LIN {X 0,Y 532.067,Z 647.363,A -85,B 0,C 180,E1 -4293.412,E2 -4293.412} C_VEL
LIN {X 0,Y 531.8,Z 656.616,A -85,B 0,C 180,E1 -4294.144,E2 -4294.144} C_VEL
LIN {X 0,Y 531.496,Z 665.466,A -85,B 0,C 180,E1 -4294.968,E2 -4294.968} C_VEL
LIN {X 0,Y 531.231,Z 673.986,A -85,B 0,C 180,E1 -4295.9,E2 -4295.9} C_VEL
LIN {X 0,Y 531.025,Z 681.116,A -85,B 0,C 180,E1 -4296.813,E2 -4296.813} C_VEL
LIN {X 0,Y 530.872,Z 687.423,A -85,B 0,C 180,E1 -4297.752,E2 -4297.752} C_VEL
LIN {X 0,Y 530.706,Z 693.662,A -85,B 0,C 180,E1 -4298.847,E2 -4298.847} C_VEL
LIN {X 0,Y 530.602,Z 698.519,A -85,B 0,C 180,E1 -4299.857,E2 -4299.857} C_VEL
LIN {X 0,Y 530.516,Z 703.385,A -85,B 0,C 180,E1 -4301.061,E2 -4301.061} C_VEL
LIN {X 0,Y 530.472,Z 707.261,A -85,B 0,C 180,E1 -4302.259,E2 -4302.259} C_VEL
LIN {X 0,Y 530.408,Z 709.397,A -85,B 0,C 180,E1 -4303.052,E2 -4303.052} C_VEL
LIN {X 0,Y 530.345,Z 712.263,A -85,B 0,C 180,E1 -4304.631,E2 -4304.631} C_VEL
LIN {X 0,Y 530.384,Z 713.236,A -85,B 0,C 180,E1 -4305.418,E2 -4305.418} C_VEL
LIN {X 0,Y 530.361,Z 713.956,A -85,B 0,C 180,E1 -4306.981,E2 -4306.981} C_VEL
LIN {X 0,Y 530.413,Z 713.28,A -85,B 0,C 180,E1 -4308.536,E2 -4308.536} C_VEL
LIN {X 0,Y 530.407,Z 712.529,A -85,B 0,C 180,E1 -4309.31,E2 -4309.31} C_VEL
LIN {X 0,Y 530.379,Z 709.752,A -85,B 0,C 180,E1 -4310.851,E2 -4310.851} C_VEL
LIN {X 0,Y 530.48,Z 706.779,A -85,B 0,C 180,E1 -4312.004,E2 -4312.004} C_VEL
LIN {X 0,Y 530.561,Z 702.949,A -85,B 0,C 180,E1 -4313.153,E2 -4313.153} C_VEL
LIN {X 0,Y 530.614,Z 698.263,A -85,B 0,C 180,E1 -4314.299,E2 -4314.299} C_VEL
LIN {X 0,Y 530.728,Z 692.661,A -85,B 0,C 180,E1 -4315.443,E2 -4315.443} C_VEL
LIN {X 0,Y 530.851,Z 685.927,A -85,B 0,C 180,E1 -4316.585,E2 -4316.585} C_VEL
LIN {X 0,Y 531.062,Z 679.305,A -85,B 0,C 180,E1 -4317.535,E2 -4317.535} C_VEL
LIN {X 0,Y 531.334,Z 671.548,A -85,B 0,C 180,E1 -4318.484,E2 -4318.484} C_VEL
LIN {X 0,Y 531.547,Z 662.423,A -85,B 0,C 180,E1 -4319.432,E2 -4319.432} C_VEL
LIN {X 0,Y 531.931,Z 652.624,A -85,B 0,C 180,E1 -4320.284,E2 -4320.284} C_VEL
LIN {X 0,Y 532.218,Z 642.253,A -85,B 0,C 180,E1 -4321.041,E2 -4321.041} C_VEL
LIN {X 0,Y 532.579,Z 629.489,A -85,B 0,C 180,E1 -4321.796,E2 -4321.796} C_VEL
LIN {X 0,Y 532.858,Z 615.986,A -85,B 0,C 180,E1 -4322.41,E2 -4322.41} C_VEL
LIN {X 0,Y 533.023,Z 602.545,A -85,B 0,C 180,E1 -4322.858,E2 -4322.858} C_VEL
LIN {X 0,Y 533.164,Z 588.82,A -85,B 0,C 180,E1 -4323.165,E2 -4323.165} C_VEL
LIN {X 0,Y 533.446,Z 541.847,A -85,B 0,C 180,E1 -4323.807,E2 -4323.807} C_VEL
LIN {X 0,Y 530.981,Z 534.347,A -85,B 0,C 180,E1 -4323.985,E2 -4323.985} C_VEL
LIN {X 0,Y 531.079,Z 534.333,A -85,B 0,C 180,E1 -4326.077,E2 -4326.077} C_VEL
LIN {X 0,Y 531.028,Z 534.337,A -85,B 0,C 180,E1 -4329.139,E2 -4329.139} C_VEL
LIN {X 0,Y 531.038,Z 534.335,A -85,B 0,C 180,E1 -4332.225,E2 -4332.225} C_VEL
LIN {X 0,Y 530.992,Z 534.346,A -85,B 0,C 180,E1 -4335.35,E2 -4335.35} C_VEL
LIN {X 0,Y 530.988,Z 534.339,A -85,B 0,C 180,E1 -4338.522,E2 -4338.522} C_VEL
LIN {X 0,Y 530.997,Z 534.34,A -85,B 0,C 180,E1 -4340.938,E2 -4340.938} C_VEL
LIN {X 0,Y 530.978,Z 534.34,A -85,B 0,C 180,E1 -4344.225,E2 -4344.225} C_VEL
LIN {X 0,Y 531.01,Z 534.336,A -85,B 0,C 180,E1 -4346.744,E2 -4346.744} C_VEL
LIN {X 0,Y 530.991,Z 534.345,A -85,B 0,C 180,E1 -4349.322,E2 -4349.322} C_VEL
LIN {X 0,Y 530.978,Z 534.337,A -85,B 0,C 180,E1 -4352.104,E2 -4352.104} C_VEL
LIN {X 0,Y 530.98,Z 534.339,A -85,B 0,C 180,E1 -4354.854,E2 -4354.854} C_VEL
LIN {X 0,Y 530.965,Z 534.346,A -85,B 0,C 180,E1 -4357.508,E2 -4357.508} C_VEL
LIN {X 0,Y 530.984,Z 534.339,A -85,B 0,C 180,E1 -4360.433,E2 -4360.433} C_VEL
LIN {X 0,Y 530.97,Z 534.348,A -85,B 0,C 180,E1 -4363.283,E2 -4363.283} C_VEL
LIN {X 0,Y 530.987,Z 534.341,A -85,B 0,C 180,E1 -4365.621,E2 -4365.621} C_VEL
LIN {X 0,Y 530.996,Z 534.338,A -85,B 0,C 180,E1 -4368.565,E2 -4368.565} C_VEL
LIN {X 0,Y 530.959,Z 534.346,A -85,B 0,C 180,E1 -4371.53,E2 -4371.53} C_VEL
LIN {X 0,Y 530.978,Z 534.343,A -85,B 0,C 180,E1 -4374.382,E2 -4374.382} C_VEL
LIN {X 0,Y 531.031,Z 534.438,A -85,B 0,C 180,E1 -4377.565,E2 -4377.565} C_VEL
LIN {X 0,Y 533.392,Z 545.862,A -85,B 0,C 180,E1 -4379.518,E2 -4379.518} C_VEL
LIN {X 0,Y 533.092,Z 562.113,A -85,B 0,C 180,E1 -4382.043,E2 -4382.043} C_VEL
LIN {X 0,Y 532.635,Z 581.906,A -85,B 0,C 180,E1 -4385.025,E2 -4385.025} C_VEL
LIN {X 0,Y 532.253,Z 602.681,A -85,B 0,C 180,E1 -4388.101,E2 -4388.101} C_VEL
LIN {X 0,Y 531.882,Z 623.757,A -85,B 0,C 180,E1 -4391.112,E2 -4391.112} C_VEL
LIN {X 0,Y 531.506,Z 643.326,A -85,B 0,C 180,E1 -4393.879,E2 -4393.879} C_VEL
LIN {X 0,Y 531.467,Z 651.526,A -85,B 0,C 180,E1 -4395.048,E2 -4395.048} C_VEL
LIN {X 0,Y 532.806,Z 661.786,A -85,B 0,C 180,E1 -4395.227,E2 -4395.227} C_VEL
LIN {X 0,Y 532.44,Z 759.968,A -85,B 0,C 180,E1 -4396.572,E2 -4396.572} C_VEL
LIN {X 0,Y 532.23,Z 773.227,A -85,B 0,C 180,E1 -4396.907,E2 -4396.907} C_VEL
LIN {X 0,Y 531.99,Z 785.378,A -85,B 0,C 180,E1 -4397.362,E2 -4397.362} C_VEL
LIN {X 0,Y 531.828,Z 796.691,A -85,B 0,C 180,E1 -4397.932,E2 -4397.932} C_VEL
LIN {X 0,Y 531.572,Z 807.906,A -85,B 0,C 180,E1 -4398.659,E2 -4398.659} C_VEL
LIN {X 0,Y 531.282,Z 818.538,A -85,B 0,C 180,E1 -4399.521,E2 -4399.521} C_VEL
LIN {X 0,Y 531.06,Z 828.119,A -85,B 0,C 180,E1 -4400.479,E2 -4400.479} C_VEL
LIN {X 0,Y 530.886,Z 835.964,A -85,B 0,C 180,E1 -4401.436,E2 -4401.436} C_VEL
LIN {X 0,Y 530.685,Z 843.624,A -85,B 0,C 180,E1 -4402.582,E2 -4402.582} C_VEL
LIN {X 0,Y 530.604,Z 850.682,A -85,B 0,C 180,E1 -4403.918,E2 -4403.918} C_VEL
LIN {X 0,Y 530.459,Z 855.372,A -85,B 0,C 180,E1 -4405.06,E2 -4405.06} C_VEL
LIN {X 0,Y 530.516,Z 858.961,A -85,B 0,C 180,E1 -4406.203,E2 -4406.203} C_VEL
LIN {X 0,Y 530.457,Z 860.811,A -85,B 0,C 180,E1 -4406.963,E2 -4406.963} C_VEL
LIN {X 0,Y 530.41,Z 862.199,A -85,B 0,C 180,E1 -4407.722,E2 -4407.722} C_VEL
LIN {X 0,Y 530.344,Z 863.787,A -85,B 0,C 180,E1 -4409.241,E2 -4409.241} C_VEL
LIN {X 0,Y 530.342,Z 864,A -85,B 0,C 180,E1 -4410,E2 -4410} C_VEL
LIN {X 0,Y 530.361,Z 863.183,A -85,B 0,C 180,E1 -4411.519,E2 -4411.519} C_VEL
LIN {X 0,Y 530.41,Z 862.195,A -85,B 0,C 180,E1 -4412.279,E2 -4412.279} C_VEL
LIN {X 0,Y 530.457,Z 860.807,A -85,B 0,C 180,E1 -4413.038,E2 -4413.038} C_VEL
LIN {X 0,Y 530.523,Z 857.895,A -85,B 0,C 180,E1 -4414.179,E2 -4414.179} C_VEL
LIN {X 0,Y 530.525,Z 853.948,A -85,B 0,C 180,E1 -4415.321,E2 -4415.321} C_VEL
LIN {X 0,Y 530.6,Z 848.259,A -85,B 0,C 180,E1 -4416.582,E2 -4416.582} C_VEL
LIN {X 0,Y 530.759,Z 841.231,A -85,B 0,C 180,E1 -4417.801,E2 -4417.801} C_VEL
LIN {X 0,Y 530.929,Z 832.99,A -85,B 0,C 180,E1 -4418.948,E2 -4418.948} C_VEL
LIN {X 0,Y 531.137,Z 824.534,A -85,B 0,C 180,E1 -4419.905,E2 -4419.905} C_VEL
LIN {X 0,Y 531.409,Z 814.088,A -85,B 0,C 180,E1 -4420.863,E2 -4420.863} C_VEL
LIN {X 0,Y 531.694,Z 803.35,A -85,B 0,C 180,E1 -4421.656,E2 -4421.656} C_VEL
LIN {X 0,Y 531.933,Z 792.394,A -85,B 0,C 180,E1 -4422.301,E2 -4422.301} C_VEL
LIN {X 0,Y 532.124,Z 780.764,A -85,B 0,C 180,E1 -4422.83,E2 -4422.83} C_VEL
LIN {X 0,Y 532.369,Z 767.341,A -85,B 0,C 180,E1 -4423.261,E2 -4423.261} C_VEL
LIN {X 0,Y 532.479,Z 754.056,A -85,B 0,C 180,E1 -4423.525,E2 -4423.525} C_VEL
LIN {X 0,Y 532.679,Z 659.294,A -85,B 0,C 180,E1 -4424.811,E2 -4424.811} C_VEL
LIN {X 0,Y 531.429,Z 651.372,A -85,B 0,C 180,E1 -4424.973,E2 -4424.973} C_VEL
LIN {X 0,Y 531.691,Z 634.591,A -85,B 0,C 180,E1 -4427.302,E2 -4427.302} C_VEL
LIN {X 0,Y 531.965,Z 611.61,A -85,B 0,C 180,E1 -4430.357,E2 -4430.357} C_VEL
LIN {X 0,Y 532.115,Z 589.217,A -85,B 0,C 180,E1 -4433.343,E2 -4433.343} C_VEL
LIN {X 0,Y 532.194,Z 568.689,A -85,B 0,C 180,E1 -4436.104,E2 -4436.104} C_VEL
LIN {X 0,Y 532.152,Z 547.238,A -85,B 0,C 180,E1 -4439.036,E2 -4439.036} C_VEL
LIN {X 0,Y 531.969,Z 539.363,A -85,B 0,C 180,E1 -4440.135,E2 -4440.135} C_VEL
LIN {X 0,Y 531.066,Z 534.337,A -85,B 0,C 180,E1 -4440.876,E2 -4440.876} C_VEL
LIN {X 0,Y 530.994,Z 534.339,A -85,B 0,C 180,E1 -4443.773,E2 -4443.773} C_VEL
LIN {X 0,Y 530.96,Z 534.346,A -85,B 0,C 180,E1 -4446.559,E2 -4446.559} C_VEL
LIN {X 0,Y 530.993,Z 534.339,A -85,B 0,C 180,E1 -4449.443,E2 -4449.443} C_VEL
LIN {X 0,Y 530.982,Z 534.343,A -85,B 0,C 180,E1 -4452.457,E2 -4452.457} C_VEL
LIN {X 0,Y 530.989,Z 534.339,A -85,B 0,C 180,E1 -4455.621,E2 -4455.621} C_VEL
LIN {X 0,Y 531.004,Z 534.343,A -85,B 0,C 180,E1 -4458.565,E2 -4458.565} C_VEL
LIN {X 0,Y 530.963,Z 534.342,A -85,B 0,C 180,E1 -4461.529,E2 -4461.529} C_VEL
LIN {X 0,Y 530.958,Z 534.348,A -85,B 0,C 180,E1 -4464.38,E2 -4464.38} C_VEL
LIN {X 0,Y 530.972,Z 534.343,A -85,B 0,C 180,E1 -4467.133,E2 -4467.133} C_VEL
LIN {X 0,Y 530.975,Z 534.341,A -85,B 0,C 180,E1 -4469.803,E2 -4469.803} C_VEL
LIN {X 0,Y 531.02,Z 534.344,A -85,B 0,C 180,E1 -4472.467,E2 -4472.467} C_VEL
LIN {X 0,Y 531.011,Z 534.34,A -85,B 0,C 180,E1 -4474.942,E2 -4474.942} C_VEL
LIN {X 0,Y 530.976,Z 534.348,A -85,B 0,C 180,E1 -4478.247,E2 -4478.247} C_VEL
LIN {X 0,Y 530.997,Z 534.344,A -85,B 0,C 180,E1 -4480.677,E2 -4480.677} C_VEL
LIN {X 0,Y 530.989,Z 534.343,A -85,B 0,C 180,E1 -4483.071,E2 -4483.071} C_VEL
LIN {X 0,Y 531.008,Z 534.343,A -85,B 0,C 180,E1 -4483.909,E2 -4483.909} C_VEL
LIN {X 0,Y 533.706,Z 542.632,A -85,B 0,C 180,E1 -4484.1,E2 -4484.1} C_VEL
LIN {X 0,Y 533.706,Z 575.669,A -85,B 0,C 180,E1 -4484.567,E2 -4484.567} C_VEL
LIN {X 0,Y 533.593,Z 590.426,A -85,B 0,C 180,E1 -4484.922,E2 -4484.922} C_VEL
LIN {X 0,Y 533.401,Z 605.575,A -85,B 0,C 180,E1 -4485.453,E2 -4485.453} C_VEL
LIN {X 0,Y 533.186,Z 619.098,A -85,B 0,C 180,E1 -4486.08,E2 -4486.08} C_VEL
LIN {X 0,Y 532.874,Z 632.267,A -85,B 0,C 180,E1 -4486.849,E2 -4486.849} C_VEL
LIN {X 0,Y 532.525,Z 645.552,A -85,B 0,C 180,E1 -4487.809,E2 -4487.809} C_VEL
LIN {X 0,Y 532.166,Z 656.516,A -85,B 0,C 180,E1 -4488.767,E2 -4488.767} C_VEL
LIN {X 0,Y 531.754,Z 667.507,A -85,B 0,C 180,E1 -4489.914,E2 -4489.914} C_VEL
LIN {X 0,Y 531.474,Z 678.111,A -85,B 0,C 180,E1 -4491.253,E2 -4491.253} C_VEL
LIN {X 0,Y 531.166,Z 686.976,A -85,B 0,C 180,E1 -4492.607,E2 -4492.607} C_VEL
LIN {X 0,Y 530.931,Z 694.109,A -85,B 0,C 180,E1 -4493.921,E2 -4493.921} C_VEL
LIN {X 0,Y 530.786,Z 700.821,A -85,B 0,C 180,E1 -4495.443,E2 -4495.443} C_VEL
LIN {X 0,Y 530.634,Z 706.106,A -85,B 0,C 180,E1 -4496.963,E2 -4496.963} C_VEL
LIN {X 0,Y 530.493,Z 710.087,A -85,B 0,C 180,E1 -4498.481,E2 -4498.481} C_VEL
LIN {X 0,Y 530.443,Z 712.856,A -85,B 0,C 180,E1 -4500,E2 -4500} C_VEL
LIN {X 0,Y 530.435,Z 714.511,A -85,B 0,C 180,E1 -4501.518,E2 -4501.518} C_VEL
LIN {X 0,Y 530.513,Z 715.05,A -85,B 0,C 180,E1 -4503.037,E2 -4503.037} C_VEL
LIN {X 0,Y 530.479,Z 714.496,A -85,B 0,C 180,E1 -4504.559,E2 -4504.559} C_VEL
LIN {X 0,Y 530.524,Z 712.816,A -85,B 0,C 180,E1 -4506.083,E2 -4506.083} C_VEL
LIN {X 0,Y 530.542,Z 709.983,A -85,B 0,C 180,E1 -4507.612,E2 -4507.612} C_VEL
LIN {X 0,Y 530.625,Z 705.935,A -85,B 0,C 180,E1 -4509.145,E2 -4509.145} C_VEL
LIN {X 0,Y 530.718,Z 700.563,A -85,B 0,C 180,E1 -4510.684,E2 -4510.684} C_VEL
LIN {X 0,Y 530.931,Z 693.643,A -85,B 0,C 180,E1 -4512.227,E2 -4512.227} C_VEL
LIN {X 0,Y 531.132,Z 686.185,A -85,B 0,C 180,E1 -4513.584,E2 -4513.584} C_VEL
LIN {X 0,Y 531.431,Z 677.07,A -85,B 0,C 180,E1 -4514.955,E2 -4514.955} C_VEL
LIN {X 0,Y 531.751,Z 667.862,A -85,B 0,C 180,E1 -4516.114,E2 -4516.114} C_VEL
LIN {X 0,Y 532.112,Z 656.77,A -85,B 0,C 180,E1 -4517.288,E2 -4517.288} C_VEL
LIN {X 0,Y 532.49,Z 644.845,A -85,B 0,C 180,E1 -4518.337,E2 -4518.337} C_VEL
LIN {X 0,Y 532.873,Z 632.308,A -85,B 0,C 180,E1 -4519.252,E2 -4519.252} C_VEL
LIN {X 0,Y 533.235,Z 619.083,A -85,B 0,C 180,E1 -4520.04,E2 -4520.04} C_VEL
LIN {X 0,Y 533.584,Z 604.796,A -85,B 0,C 180,E1 -4520.715,E2 -4520.715} C_VEL
LIN {X 0,Y 533.819,Z 588.996,A -85,B 0,C 180,E1 -4521.276,E2 -4521.276} C_VEL
LIN {X 0,Y 533.987,Z 573.698,A -85,B 0,C 180,E1 -4521.65,E2 -4521.65} C_VEL
LIN {X 0,Y 534.035,Z 542.955,A -85,B 0,C 180,E1 -4522.104,E2 -4522.104} C_VEL
LIN {X 0,Y 530.951,Z 534.348,A -85,B 0,C 180,E1 -4522.338,E2 -4522.338} C_VEL
LIN {X 0,Y 530.996,Z 534.338,A -85,B 0,C 180,E1 -4525.058,E2 -4525.058} C_VEL
LIN {X 0,Y 531.017,Z 534.338,A -85,B 0,C 180,E1 -4527.595,E2 -4527.595} C_VEL
LIN {X 0,Y 530.975,Z 534.34,A -85,B 0,C 180,E1 -4530.645,E2 -4530.645} C_VEL
LIN {X 0,Y 530.988,Z 534.341,A -85,B 0,C 180,E1 -4533.772,E2 -4533.772} C_VEL
LIN {X 0,Y 530.97,Z 534.341,A -85,B 0,C 180,E1 -4534.128,E2 -4534.128} C_VEL
LIN {X 0,Y 530.296,Z 534.425,A -85,B 0,C 180,E1 -4534.761,E2 -4534.761} C_VEL
LIN {X 0,Y 527.427,Z 534.785,A -85,B 0,C 180,E1 -4535.789,E2 -4535.789} C_VEL
LIN {X 0,Y 525.01,Z 535.085,A -85,B 0,C 180,E1 -4536.617,E2 -4536.617} C_VEL
LIN {X 0,Y 523.982,Z 535.21,A -85,B 0,C 180,E1 -4537.257,E2 -4537.257} C_VEL
LIN {X 0,Y 523.904,Z 535.22,A -85,B 0,C 180,E1 -4537.473,E2 -4537.473} C_VEL
LIN {X 0,Y 523.938,Z 535.223,A -85,B 0,C 180,E1 -4540.129,E2 -4540.129} C_VEL
LIN {X 0,Y 523.938,Z 535.222,A -85,B 0,C 180,E1 -4542.459,E2 -4542.459} C_VEL
LIN {X 0,Y 523.946,Z 535.214,A -85,B 0,C 180,E1 -4545.309,E2 -4545.309} C_VEL
LIN {X 0,Y 523.958,Z 535.217,A -85,B 0,C 180,E1 -4548.689,E2 -4548.689} C_VEL
LIN {X 0,Y 523.919,Z 535.219,A -85,B 0,C 180,E1 -4551.08,E2 -4551.08} C_VEL
LIN {X 0,Y 523.905,Z 535.22,A -85,B 0,C 180,E1 -4553.825,E2 -4553.825} C_VEL
LIN {X 0,Y 523.942,Z 535.223,A -85,B 0,C 180,E1 -4556.635,E2 -4556.635} C_VEL
LIN {X 0,Y 523.956,Z 535.213,A -85,B 0,C 180,E1 -4559.355,E2 -4559.355} C_VEL
LIN {X 0,Y 523.978,Z 535.214,A -85,B 0,C 180,E1 -4562.281,E2 -4562.281} C_VEL
LIN {X 0,Y 523.953,Z 535.222,A -85,B 0,C 180,E1 -4564.581,E2 -4564.581} C_VEL
LIN {X 0,Y 523.916,Z 535.222,A -85,B 0,C 180,E1 -4567.106,E2 -4567.106} C_VEL
LIN {X 0,Y 523.978,Z 535.21,A -85,B 0,C 180,E1 -4569.865,E2 -4569.865} C_VEL
LIN {X 0,Y 523.966,Z 535.222,A -85,B 0,C 180,E1 -4572.837,E2 -4572.837} C_VEL
LIN {X 0,Y 523.976,Z 535.214,A -85,B 0,C 180,E1 -4575.235,E2 -4575.235} C_VEL
LIN {X 0,Y 524.011,Z 535.208,A -85,B 0,C 180,E1 -4578.394,E2 -4578.394} C_VEL
LIN {X 0,Y 524.004,Z 535.209,A -85,B 0,C 180,E1 -4581.516,E2 -4581.516} C_VEL
LIN {X 0,Y 524.081,Z 535.201,A -85,B 0,C 180,E1 -4584.613,E2 -4584.613} C_VEL
LIN {X 0,Y 524.111,Z 535.195,A -85,B 0,C 180,E1 -4587.694,E2 -4587.694} C_VEL
LIN {X 0,Y 524.121,Z 535.196,A -85,B 0,C 180,E1 -4590.768,E2 -4590.768} C_VEL
LIN {X 0,Y 524.072,Z 535.206,A -85,B 0,C 180,E1 -4593.074,E2 -4593.074} C_VEL
LIN {X 0,Y 524.035,Z 535.203,A -85,B 0,C 180,E1 -4596.159,E2 -4596.159} C_VEL
LIN {X 0,Y 524.002,Z 535.207,A -85,B 0,C 180,E1 -4598.484,E2 -4598.484} C_VEL
LIN {X 0,Y 524.022,Z 535.208,A -85,B 0,C 180,E1 -4601.751,E2 -4601.751} C_VEL
LIN {X 0,Y 523.99,Z 535.213,A -85,B 0,C 180,E1 -4605.052,E2 -4605.052} C_VEL
LIN {X 0,Y 523.961,Z 535.215,A -85,B 0,C 180,E1 -4607.969,E2 -4607.969} C_VEL
LIN {X 0,Y 523.969,Z 535.211,A -85,B 0,C 180,E1 -4610.41,E2 -4610.41} C_VEL
LIN {X 0,Y 523.914,Z 535.219,A -85,B 0,C 180,E1 -4612.893,E2 -4612.893} C_VEL
LIN {X 0,Y 523.952,Z 535.22,A -85,B 0,C 180,E1 -4615.418,E2 -4615.418} C_VEL
LIN {X 0,Y 523.967,Z 535.216,A -85,B 0,C 180,E1 -4617.998,E2 -4617.998} C_VEL
LIN {X 0,Y 523.949,Z 535.214,A -85,B 0,C 180,E1 -4620.856,E2 -4620.856} C_VEL
LIN {X 0,Y 523.959,Z 535.222,A -85,B 0,C 180,E1 -4623.735,E2 -4623.735} C_VEL
LIN {X 0,Y 523.918,Z 535.219,A -85,B 0,C 180,E1 -4626.404,E2 -4626.404} C_VEL
LIN {X 0,Y 523.927,Z 535.217,A -85,B 0,C 180,E1 -4629.083,E2 -4629.083} C_VEL
LIN {X 0,Y 523.952,Z 535.22,A -85,B 0,C 180,E1 -4632.118,E2 -4632.118} C_VEL
LIN {X 0,Y 523.951,Z 535.215,A -85,B 0,C 180,E1 -4635.308,E2 -4635.308} C_VEL
LIN {X 0,Y 523.968,Z 535.213,A -85,B 0,C 180,E1 -4638.687,E2 -4638.687} C_VEL
LIN {X 0,Y 523.949,Z 535.214,A -85,B 0,C 180,E1 -4641.075,E2 -4641.075} C_VEL
LIN {X 0,Y 523.925,Z 535.222,A -85,B 0,C 180,E1 -4643.828,E2 -4643.828} C_VEL
LIN {X 0,Y 523.939,Z 535.219,A -85,B 0,C 180,E1 -4646.636,E2 -4646.636} C_VEL
LIN {X 0,Y 524,Z 535.362,A -85,B 0,C 180,E1 -4649.872,E2 -4649.872} C_VEL
LIN {X 0,Y 526.576,Z 542.941,A -85,B 0,C 180,E1 -4650.059,E2 -4650.059} C_VEL
LIN {X 0,Y 526.347,Z 592.723,A -85,B 0,C 180,E1 -4650.778,E2 -4650.778} C_VEL
LIN {X 0,Y 526.142,Z 606.279,A -85,B 0,C 180,E1 -4651.121,E2 -4651.121} C_VEL
LIN {X 0,Y 525.954,Z 619.038,A -85,B 0,C 180,E1 -4651.588,E2 -4651.588} C_VEL
LIN {X 0,Y 525.701,Z 630.952,A -85,B 0,C 180,E1 -4652.156,E2 -4652.156} C_VEL
LIN {X 0,Y 525.293,Z 644.038,A -85,B 0,C 180,E1 -4652.942,E2 -4652.942} C_VEL
LIN {X 0,Y 524.985,Z 656.089,A -85,B 0,C 180,E1 -4653.864,E2 -4653.864} C_VEL
LIN {X 0,Y 524.6,Z 666.43,A -85,B 0,C 180,E1 -4654.828,E2 -4654.828} C_VEL
LIN {X 0,Y 524.294,Z 675.348,A -85,B 0,C 180,E1 -4655.818,E2 -4655.818} C_VEL
LIN {X 0,Y 524.059,Z 683.564,A -85,B 0,C 180,E1 -4656.905,E2 -4656.905} C_VEL
LIN {X 0,Y 523.847,Z 691.372,A -85,B 0,C 180,E1 -4658.143,E2 -4658.143} C_VEL
LIN {X 0,Y 523.623,Z 698.674,A -85,B 0,C 180,E1 -4659.576,E2 -4659.576} C_VEL
LIN {X 0,Y 523.534,Z 703.615,A -85,B 0,C 180,E1 -4660.799,E2 -4660.799} C_VEL
LIN {X 0,Y 523.451,Z 707.521,A -85,B 0,C 180,E1 -4662.013,E2 -4662.013} C_VEL
LIN {X 0,Y 523.392,Z 709.617,A -85,B 0,C 180,E1 -4662.818,E2 -4662.818} C_VEL
LIN {X 0,Y 523.282,Z 712.651,A -85,B 0,C 180,E1 -4664.419,E2 -4664.419} C_VEL
LIN {X 0,Y 523.325,Z 714.167,A -85,B 0,C 180,E1 -4666.012,E2 -4666.012} C_VEL
LIN {X 0,Y 523.288,Z 714.519,A -85,B 0,C 180,E1 -4666.802,E2 -4666.802} C_VEL
LIN {X 0,Y 523.355,Z 713.806,A -85,B 0,C 180,E1 -4668.604,E2 -4668.604} C_VEL
LIN {X 0,Y 523.338,Z 712.204,A -85,B 0,C 180,E1 -4669.946,E2 -4669.946} C_VEL
LIN {X 0,Y 523.334,Z 710.858,A -85,B 0,C 180,E1 -4670.727,E2 -4670.727} C_VEL
LIN {X 0,Y 523.455,Z 706.94,A -85,B 0,C 180,E1 -4672.284,E2 -4672.284} C_VEL
LIN {X 0,Y 523.564,Z 703.351,A -85,B 0,C 180,E1 -4673.373,E2 -4673.373} C_VEL
LIN {X 0,Y 523.618,Z 698.295,A -85,B 0,C 180,E1 -4674.609,E2 -4674.609} C_VEL
LIN {X 0,Y 523.792,Z 692.471,A -85,B 0,C 180,E1 -4675.768,E2 -4675.768} C_VEL
LIN {X 0,Y 523.985,Z 685.49,A -85,B 0,C 180,E1 -4676.925,E2 -4676.925} C_VEL
LIN {X 0,Y 524.29,Z 677.121,A -85,B 0,C 180,E1 -4678.08,E2 -4678.08} C_VEL
LIN {X 0,Y 524.563,Z 667.007,A -85,B 0,C 180,E1 -4679.233,E2 -4679.233} C_VEL
LIN {X 0,Y 524.958,Z 656.704,A -85,B 0,C 180,E1 -4680.192,E2 -4680.192} C_VEL
LIN {X 0,Y 525.321,Z 645.456,A -85,B 0,C 180,E1 -4681.054,E2 -4681.054} C_VEL
LIN {X 0,Y 525.585,Z 634.848,A -85,B 0,C 180,E1 -4681.724,E2 -4681.724} C_VEL
LIN {X 0,Y 525.918,Z 621.553,A -85,B 0,C 180,E1 -4682.394,E2 -4682.394} C_VEL
LIN {X 0,Y 526.154,Z 606.681,A -85,B 0,C 180,E1 -4682.943,E2 -4682.943} C_VEL
LIN {X 0,Y 526.238,Z 592.192,A -85,B 0,C 180,E1 -4683.302,E2 -4683.302} C_VEL
LIN {X 0,Y 526.49,Z 542.929,A -85,B 0,C 180,E1 -4683.995,E2 -4683.995} C_VEL
LIN {X 0,Y 523.965,Z 535.219,A -85,B 0,C 180,E1 -4684.183,E2 -4684.183} C_VEL
LIN {X 0,Y 524.042,Z 535.209,A -85,B 0,C 180,E1 -4686.159,E2 -4686.159} C_VEL
LIN {X 0,Y 523.996,Z 535.215,A -85,B 0,C 180,E1 -4689.262,E2 -4689.262} C_VEL
LIN {X 0,Y 524.022,Z 535.214,A -85,B 0,C 180,E1 -4691.752,E2 -4691.752} C_VEL
LIN {X 0,Y 523.99,Z 535.215,A -85,B 0,C 180,E1 -4695.053,E2 -4695.053} C_VEL
LIN {X 0,Y 523.961,Z 535.218,A -85,B 0,C 180,E1 -4697.969,E2 -4697.969} C_VEL
LIN {X 0,Y 523.969,Z 535.214,A -85,B 0,C 180,E1 -4700.41,E2 -4700.41} C_VEL
LIN {X 0,Y 523.915,Z 535.222,A -85,B 0,C 180,E1 -4702.894,E2 -4702.894} C_VEL
LIN {X 0,Y 523.953,Z 535.221,A -85,B 0,C 180,E1 -4705.419,E2 -4705.419} C_VEL
LIN {X 0,Y 523.969,Z 535.213,A -85,B 0,C 180,E1 -4707.999,E2 -4707.999} C_VEL
LIN {X 0,Y 523.951,Z 535.215,A -85,B 0,C 180,E1 -4710.857,E2 -4710.857} C_VEL
LIN {X 0,Y 523.959,Z 535.214,A -85,B 0,C 180,E1 -4713.735,E2 -4713.735} C_VEL
LIN {X 0,Y 523.906,Z 535.219,A -85,B 0,C 180,E1 -4716.403,E2 -4716.403} C_VEL
LIN {X 0,Y 523.923,Z 535.224,A -85,B 0,C 180,E1 -4719.085,E2 -4719.085} C_VEL
LIN {X 0,Y 523.957,Z 535.213,A -85,B 0,C 180,E1 -4722.119,E2 -4722.119} C_VEL
LIN {X 0,Y 523.955,Z 535.221,A -85,B 0,C 180,E1 -4725.309,E2 -4725.309} C_VEL
LIN {X 0,Y 523.958,Z 535.216,A -85,B 0,C 180,E1 -4728.69,E2 -4728.69} C_VEL
LIN {X 0,Y 523.917,Z 535.221,A -85,B 0,C 180,E1 -4731.899,E2 -4731.899} C_VEL
LIN {X 0,Y 523.937,Z 535.225,A -85,B 0,C 180,E1 -4734.91,E2 -4734.91} C_VEL
LIN {X 0,Y 523.998,Z 535.338,A -85,B 0,C 180,E1 -4737.328,E2 -4737.328} C_VEL
LIN {X 0,Y 526.441,Z 546.745,A -85,B 0,C 180,E1 -4739.317,E2 -4739.317} C_VEL
LIN {X 0,Y 526.306,Z 557.642,A -85,B 0,C 180,E1 -4741.05,E2 -4741.05} C_VEL
LIN {X 0,Y 525.818,Z 575.623,A -85,B 0,C 180,E1 -4743.828,E2 -4743.828} C_VEL
LIN {X 0,Y 525.423,Z 595.021,A -85,B 0,C 180,E1 -4746.76,E2 -4746.76} C_VEL
LIN {X 0,Y 525.04,Z 614.456,A -85,B 0,C 180,E1 -4749.634,E2 -4749.634} C_VEL
LIN {X 0,Y 524.636,Z 635.502,A -85,B 0,C 180,E1 -4752.659,E2 -4752.659} C_VEL
LIN {X 0,Y 524.408,Z 650.562,A -85,B 0,C 180,E1 -4754.813,E2 -4754.813} C_VEL
LIN {X 0,Y 525.98,Z 662.858,A -85,B 0,C 180,E1 -4755.039,E2 -4755.039} C_VEL
LIN {X 0,Y 525.538,Z 758.417,A -85,B 0,C 180,E1 -4756.368,E2 -4756.368} C_VEL
LIN {X 0,Y 525.342,Z 771.445,A -85,B 0,C 180,E1 -4756.683,E2 -4756.683} C_VEL
LIN {X 0,Y 525.041,Z 785.224,A -85,B 0,C 180,E1 -4757.192,E2 -4757.192} C_VEL
LIN {X 0,Y 524.874,Z 797.406,A -85,B 0,C 180,E1 -4757.813,E2 -4757.813} C_VEL
LIN {X 0,Y 524.555,Z 809.196,A -85,B 0,C 180,E1 -4758.603,E2 -4758.603} C_VEL
LIN {X 0,Y 524.241,Z 819.606,A -85,B 0,C 180,E1 -4759.476,E2 -4759.476} C_VEL
LIN {X 0,Y 524.054,Z 828.119,A -85,B 0,C 180,E1 -4760.35,E2 -4760.35} C_VEL
LIN {X 0,Y 523.852,Z 835.964,A -85,B 0,C 180,E1 -4761.32,E2 -4761.32} C_VEL
LIN {X 0,Y 523.633,Z 843.624,A -85,B 0,C 180,E1 -4762.481,E2 -4762.481} C_VEL
LIN {X 0,Y 523.515,Z 850.682,A -85,B 0,C 180,E1 -4763.835,E2 -4763.835} C_VEL
LIN {X 0,Y 523.384,Z 855.372,A -85,B 0,C 180,E1 -4764.993,E2 -4764.993} C_VEL
LIN {X 0,Y 523.443,Z 858.96,A -85,B 0,C 180,E1 -4766.151,E2 -4766.151} C_VEL
LIN {X 0,Y 523.368,Z 860.811,A -85,B 0,C 180,E1 -4766.921,E2 -4766.921} C_VEL
LIN {X 0,Y 523.334,Z 862.198,A -85,B 0,C 180,E1 -4767.692,E2 -4767.692} C_VEL
LIN {X 0,Y 523.25,Z 863.787,A -85,B 0,C 180,E1 -4769.231,E2 -4769.231} C_VEL
LIN {X 0,Y 523.246,Z 864,A -85,B 0,C 180,E1 -4770,E2 -4770} C_VEL
LIN {X 0,Y 523.274,Z 863.182,A -85,B 0,C 180,E1 -4771.54,E2 -4771.54} C_VEL
LIN {X 0,Y 523.334,Z 862.194,A -85,B 0,C 180,E1 -4772.309,E2 -4772.309} C_VEL
LIN {X 0,Y 523.368,Z 860.807,A -85,B 0,C 180,E1 -4773.079,E2 -4773.079} C_VEL
LIN {X 0,Y 523.442,Z 857.895,A -85,B 0,C 180,E1 -4774.235,E2 -4774.235} C_VEL
LIN {X 0,Y 523.464,Z 853.948,A -85,B 0,C 180,E1 -4775.393,E2 -4775.393} C_VEL
LIN {X 0,Y 523.524,Z 848.724,A -85,B 0,C 180,E1 -4776.581,E2 -4776.581} C_VEL
LIN {X 0,Y 523.666,Z 842.458,A -85,B 0,C 180,E1 -4777.713,E2 -4777.713} C_VEL
LIN {X 0,Y 523.855,Z 834.474,A -85,B 0,C 180,E1 -4778.876,E2 -4778.876} C_VEL
LIN {X 0,Y 524.108,Z 826.328,A -85,B 0,C 180,E1 -4779.845,E2 -4779.845} C_VEL
LIN {X 0,Y 524.367,Z 816.395,A -85,B 0,C 180,E1 -4780.815,E2 -4780.815} C_VEL
LIN {X 0,Y 524.665,Z 805.175,A -85,B 0,C 180,E1 -4781.689,E2 -4781.689} C_VEL
LIN {X 0,Y 524.927,Z 794.114,A -85,B 0,C 180,E1 -4782.37,E2 -4782.37} C_VEL
LIN {X 0,Y 525.157,Z 781.764,A -85,B 0,C 180,E1 -4782.954,E2 -4782.954} C_VEL
LIN {X 0,Y 525.401,Z 768.706,A -85,B 0,C 180,E1 -4783.391,E2 -4783.391} C_VEL
LIN {X 0,Y 525.552,Z 754.891,A -85,B 0,C 180,E1 -4783.682,E2 -4783.682} C_VEL
LIN {X 0,Y 525.883,Z 660.941,A -85,B 0,C 180,E1 -4784.975,E2 -4784.975} C_VEL
LIN {X 0,Y 524.344,Z 649.901,A -85,B 0,C 180,E1 -4785.193,E2 -4785.193} C_VEL
LIN {X 0,Y 524.732,Z 626.855,A -85,B 0,C 180,E1 -4788.306,E2 -4788.306} C_VEL
LIN {X 0,Y 524.93,Z 605.416,A -85,B 0,C 180,E1 -4791.192,E2 -4791.192} C_VEL
LIN {X 0,Y 525.067,Z 584.025,A -85,B 0,C 180,E1 -4794.095,E2 -4794.095} C_VEL
LIN {X 0,Y 525.127,Z 563.905,A -85,B 0,C 180,E1 -4796.852,E2 -4796.852} C_VEL
LIN {X 0,Y 525.117,Z 543.644,A -85,B 0,C 180,E1 -4799.683,E2 -4799.683} C_VEL
LIN {X 0,Y 524.644,Z 538.85,A -85,B 0,C 180,E1 -4800.378,E2 -4800.378} C_VEL
LIN {X 0,Y 524.022,Z 535.215,A -85,B 0,C 180,E1 -4800.932,E2 -4800.932} C_VEL
LIN {X 0,Y 523.945,Z 535.219,A -85,B 0,C 180,E1 -4804.29,E2 -4804.29} C_VEL
LIN {X 0,Y 523.912,Z 535.225,A -85,B 0,C 180,E1 -4807.132,E2 -4807.132} C_VEL
LIN {X 0,Y 523.942,Z 535.216,A -85,B 0,C 180,E1 -4810.13,E2 -4810.13} C_VEL
LIN {X 0,Y 523.939,Z 535.22,A -85,B 0,C 180,E1 -4812.459,E2 -4812.459} C_VEL
LIN {X 0,Y 523.958,Z 535.216,A -85,B 0,C 180,E1 -4815.309,E2 -4815.309} C_VEL
LIN {X 0,Y 523.966,Z 535.22,A -85,B 0,C 180,E1 -4818.689,E2 -4818.689} C_VEL
LIN {X 0,Y 523.921,Z 535.219,A -85,B 0,C 180,E1 -4821.898,E2 -4821.898} C_VEL
LIN {X 0,Y 523.929,Z 535.223,A -85,B 0,C 180,E1 -4824.911,E2 -4824.911} C_VEL
LIN {X 0,Y 523.94,Z 535.217,A -85,B 0,C 180,E1 -4827.68,E2 -4827.68} C_VEL
LIN {X 0,Y 523.959,Z 535.221,A -85,B 0,C 180,E1 -4830.676,E2 -4830.676} C_VEL
LIN {X 0,Y 523.979,Z 535.214,A -85,B 0,C 180,E1 -4833.728,E2 -4833.728} C_VEL
LIN {X 0,Y 523.94,Z 535.224,A -85,B 0,C 180,E1 -4836.271,E2 -4836.271} C_VEL
LIN {X 0,Y 523.95,Z 535.221,A -85,B 0,C 180,E1 -4838.766,E2 -4838.766} C_VEL
LIN {X 0,Y 523.953,Z 535.218,A -85,B 0,C 180,E1 -4841.22,E2 -4841.22} C_VEL
LIN {X 0,Y 523.957,Z 535.22,A -85,B 0,C 180,E1 -4843.713,E2 -4843.713} C_VEL
LIN {X 0,Y 526.975,Z 544.747,A -85,B 0,C 180,E1 -4843.936,E2 -4843.936} C_VEL
LIN {X 0,Y 526.849,Z 576.935,A -85,B 0,C 180,E1 -4844.39,E2 -4844.39} C_VEL
LIN {X 0,Y 526.772,Z 591.651,A -85,B 0,C 180,E1 -4844.747,E2 -4844.747} C_VEL
LIN {X 0,Y 526.57,Z 606.323,A -85,B 0,C 180,E1 -4845.26,E2 -4845.26} C_VEL
LIN {X 0,Y 526.353,Z 619.984,A -85,B 0,C 180,E1 -4845.896,E2 -4845.896} C_VEL
LIN {X 0,Y 526.035,Z 633.256,A -85,B 0,C 180,E1 -4846.675,E2 -4846.675} C_VEL
LIN {X 0,Y 525.678,Z 646.615,A -85,B 0,C 180,E1 -4847.648,E2 -4847.648} C_VEL
LIN {X 0,Y 525.303,Z 657.603,A -85,B 0,C 180,E1 -4848.618,E2 -4848.618} C_VEL
LIN {X 0,Y 524.855,Z 668.638,A -85,B 0,C 180,E1 -4849.78,E2 -4849.78} C_VEL
LIN {X 0,Y 524.555,Z 679.265,A -85,B 0,C 180,E1 -4851.136,E2 -4851.136} C_VEL
LIN {X 0,Y 524.233,Z 688.527,A -85,B 0,C 180,E1 -4852.576,E2 -4852.576} C_VEL
LIN {X 0,Y 523.99,Z 695.25,A -85,B 0,C 180,E1 -4853.84,E2 -4853.84} C_VEL
LIN {X 0,Y 523.803,Z 701.968,A -85,B 0,C 180,E1 -4855.382,E2 -4855.382} C_VEL
LIN {X 0,Y 523.651,Z 707.229,A -85,B 0,C 180,E1 -4856.922,E2 -4856.922} C_VEL
LIN {X 0,Y 523.502,Z 711.188,A -85,B 0,C 180,E1 -4858.461,E2 -4858.461} C_VEL
LIN {X 0,Y 523.441,Z 713.941,A -85,B 0,C 180,E1 -4860,E2 -4860} C_VEL
LIN {X 0,Y 523.423,Z 715.571,A -85,B 0,C 180,E1 -4861.538,E2 -4861.538} C_VEL
LIN {X 0,Y 523.486,Z 716.072,A -85,B 0,C 180,E1 -4863.078,E2 -4863.078} C_VEL
LIN {X 0,Y 523.468,Z 715.473,A -85,B 0,C 180,E1 -4864.62,E2 -4864.62} C_VEL
LIN {X 0,Y 523.524,Z 713.74,A -85,B 0,C 180,E1 -4866.165,E2 -4866.165} C_VEL
LIN {X 0,Y 523.544,Z 710.856,A -85,B 0,C 180,E1 -4867.714,E2 -4867.714} C_VEL
LIN {X 0,Y 523.642,Z 706.751,A -85,B 0,C 180,E1 -4869.268,E2 -4869.268} C_VEL
LIN {X 0,Y 523.748,Z 701.289,A -85,B 0,C 180,E1 -4870.828,E2 -4870.828} C_VEL
LIN {X 0,Y 523.97,Z 694.293,A -85,B 0,C 180,E1 -4872.392,E2 -4872.392} C_VEL
LIN {X 0,Y 524.22,Z 686.758,A -85,B 0,C 180,E1 -4873.766,E2 -4873.766} C_VEL
LIN {X 0,Y 524.526,Z 677.899,A -85,B 0,C 180,E1 -4875.106,E2 -4875.106} C_VEL
LIN {X 0,Y 524.887,Z 668.215,A -85,B 0,C 180,E1 -4876.33,E2 -4876.33} C_VEL
LIN {X 0,Y 525.26,Z 656.961,A -85,B 0,C 180,E1 -4877.52,E2 -4877.52} C_VEL
LIN {X 0,Y 525.668,Z 645.081,A -85,B 0,C 180,E1 -4878.567,E2 -4878.567} C_VEL
LIN {X 0,Y 526.095,Z 632.119,A -85,B 0,C 180,E1 -4879.51,E2 -4879.51} C_VEL
LIN {X 0,Y 526.476,Z 618.583,A -85,B 0,C 180,E1 -4880.308,E2 -4880.308} C_VEL
LIN {X 0,Y 526.782,Z 604.921,A -85,B 0,C 180,E1 -4880.949,E2 -4880.949} C_VEL
LIN {X 0,Y 527.027,Z 589.742,A -85,B 0,C 180,E1 -4881.487,E2 -4881.487} C_VEL
LIN {X 0,Y 527.194,Z 574.247,A -85,B 0,C 180,E1 -4881.865,E2 -4881.865} C_VEL
LIN {X 0,Y 527.246,Z 544.642,A -85,B 0,C 180,E1 -4882.306,E2 -4882.306} C_VEL
LIN {X 0,Y 523.925,Z 535.222,A -85,B 0,C 180,E1 -4882.561,E2 -4882.561} C_VEL
LIN {X 0,Y 523.949,Z 535.219,A -85,B 0,C 180,E1 -4885.418,E2 -4885.418} C_VEL
LIN {X 0,Y 523.971,Z 535.221,A -85,B 0,C 180,E1 -4887.998,E2 -4887.998} C_VEL
LIN {X 0,Y 523.946,Z 535.214,A -85,B 0,C 180,E1 -4890.854,E2 -4890.854} C_VEL
LIN {X 0,Y 523.96,Z 535.216,A -85,B 0,C 180,E1 -4893.734,E2 -4893.734} C_VEL
LIN {X 0,Y 523.904,Z 535.225,A -85,B 0,C 180,E1 -4896.401,E2 -4896.401} C_VEL
LIN {X 0,Y 523.904,Z 535.22,A -85,B 0,C 180,E1 -4897.473,E2 -4897.473} C_VEL
LIN {X 0,Y 523.253,Z 535.309,A -85,B 0,C 180,E1 -4898.115,E2 -4898.115} C_VEL
LIN {X 0,Y 520.411,Z 535.662,A -85,B 0,C 180,E1 -4899.158,E2 -4899.158} C_VEL
LIN {X 0,Y 518.002,Z 535.961,A -85,B 0,C 180,E1 -4899.998,E2 -4899.998} C_VEL
LIN {X 0,Y 516.967,Z 536.088,A -85,B 0,C 180,E1 -4900.646,E2 -4900.646} C_VEL
LIN {X 0,Y 516.884,Z 536.095,A -85,B 0,C 180,E1 -4900.865,E2 -4900.865} C_VEL
LIN {X 0,Y 516.883,Z 536.098,A -85,B 0,C 180,E1 -4903.903,E2 -4903.903} C_VEL
LIN {X 0,Y 516.884,Z 536.094,A -85,B 0,C 180,E1 -4907.168,E2 -4907.168} C_VEL
LIN {X 0,Y 516.885,Z 536.094,A -85,B 0,C 180,E1 -4909.589,E2 -4909.589} C_VEL
LIN {X 0,Y 516.864,Z 536.103,A -85,B 0,C 180,E1 -4912.274,E2 -4912.274} C_VEL
LIN {X 0,Y 516.89,Z 536.094,A -85,B 0,C 180,E1 -4915.175,E2 -4915.175} C_VEL
LIN {X 0,Y 516.876,Z 536.096,A -85,B 0,C 180,E1 -4917.975,E2 -4917.975} C_VEL
LIN {X 0,Y 516.921,Z 536.098,A -85,B 0,C 180,E1 -4920.695,E2 -4920.695} C_VEL
LIN {X 0,Y 516.942,Z 536.087,A -85,B 0,C 180,E1 -4923.803,E2 -4923.803} C_VEL
LIN {X 0,Y 516.872,Z 536.104,A -85,B 0,C 180,E1 -4926.776,E2 -4926.776} C_VEL
LIN {X 0,Y 516.939,Z 536.087,A -85,B 0,C 180,E1 -4929.731,E2 -4929.731} C_VEL
LIN {X 0,Y 516.928,Z 536.094,A -85,B 0,C 180,E1 -4932.596,E2 -4932.596} C_VEL
LIN {X 0,Y 516.941,Z 536.094,A -85,B 0,C 180,E1 -4935.03,E2 -4935.03} C_VEL
LIN {X 0,Y 516.964,Z 536.085,A -85,B 0,C 180,E1 -4938.233,E2 -4938.233} C_VEL
LIN {X 0,Y 516.969,Z 536.087,A -85,B 0,C 180,E1 -4941.399,E2 -4941.399} C_VEL
LIN {X 0,Y 517.009,Z 536.079,A -85,B 0,C 180,E1 -4943.756,E2 -4943.756} C_VEL
LIN {X 0,Y 517.084,Z 536.071,A -85,B 0,C 180,E1 -4947.663,E2 -4947.663} C_VEL
LIN {X 0,Y 517.092,Z 536.072,A -85,B 0,C 180,E1 -4950.778,E2 -4950.778} C_VEL
LIN {X 0,Y 517.013,Z 536.086,A -85,B 0,C 180,E1 -4953.116,E2 -4953.116} C_VEL
LIN {X 0,Y 517.001,Z 536.079,A -85,B 0,C 180,E1 -4956.243,E2 -4956.243} C_VEL
LIN {X 0,Y 516.95,Z 536.094,A -85,B 0,C 180,E1 -4959.389,E2 -4959.389} C_VEL
LIN {X 0,Y 516.981,Z 536.085,A -85,B 0,C 180,E1 -4961.824,E2 -4961.824} C_VEL
LIN {X 0,Y 516.941,Z 536.092,A -85,B 0,C 180,E1 -4965.146,E2 -4965.146} C_VEL
LIN {X 0,Y 516.923,Z 536.09,A -85,B 0,C 180,E1 -4968.222,E2 -4968.222} C_VEL
LIN {X 0,Y 516.909,Z 536.091,A -85,B 0,C 180,E1 -4970.701,E2 -4970.701} C_VEL
LIN {X 0,Y 516.908,Z 536.094,A -85,B 0,C 180,E1 -4974.072,E2 -4974.072} C_VEL
LIN {X 0,Y 516.925,Z 536.089,A -85,B 0,C 180,E1 -4976.657,E2 -4976.657} C_VEL
LIN {X 0,Y 516.921,Z 536.096,A -85,B 0,C 180,E1 -4979.526,E2 -4979.526} C_VEL
LIN {X 0,Y 516.897,Z 536.093,A -85,B 0,C 180,E1 -4982.544,E2 -4982.544} C_VEL
LIN {X 0,Y 516.879,Z 536.097,A -85,B 0,C 180,E1 -4985.332,E2 -4985.332} C_VEL
LIN {X 0,Y 516.877,Z 536.103,A -85,B 0,C 180,E1 -4987.943,E2 -4987.943} C_VEL
LIN {X 0,Y 516.899,Z 536.092,A -85,B 0,C 180,E1 -4990.739,E2 -4990.739} C_VEL
LIN {X 0,Y 516.877,Z 536.104,A -85,B 0,C 180,E1 -4993.903,E2 -4993.903} C_VEL
LIN {X 0,Y 516.877,Z 536.103,A -85,B 0,C 180,E1 -4996.107,E2 -4996.107} C_VEL
LIN {X 0,Y 516.907,Z 536.091,A -85,B 0,C 180,E1 -4999.261,E2 -4999.261} C_VEL
LIN {X 0,Y 516.878,Z 536.104,A -85,B 0,C 180,E1 -5002.056,E2 -5002.056} C_VEL
LIN {X 0,Y 516.891,Z 536.093,A -85,B 0,C 180,E1 -5005.176,E2 -5005.176} C_VEL
LIN {X 0,Y 516.879,Z 536.102,A -85,B 0,C 180,E1 -5007.976,E2 -5007.976} C_VEL
LIN {X 0,Y 516.922,Z 536.122,A -85,B 0,C 180,E1 -5009.653,E2 -5009.653} C_VEL
LIN {X 0,Y 519.82,Z 544.628,A -85,B 0,C 180,E1 -5009.868,E2 -5009.868} C_VEL
LIN {X 0,Y 519.508,Z 593.268,A -85,B 0,C 180,E1 -5010.578,E2 -5010.578} C_VEL
LIN {X 0,Y 519.286,Z 607.774,A -85,B 0,C 180,E1 -5010.949,E2 -5010.949} C_VEL
LIN {X 0,Y 519.105,Z 620.55,A -85,B 0,C 180,E1 -5011.428,E2 -5011.428} C_VEL
LIN {X 0,Y 518.836,Z 632.838,A -85,B 0,C 180,E1 -5012.03,E2 -5012.03} C_VEL
LIN {X 0,Y 518.446,Z 644.935,A -85,B 0,C 180,E1 -5012.774,E2 -5012.774} C_VEL
LIN {X 0,Y 518.128,Z 656.332,A -85,B 0,C 180,E1 -5013.646,E2 -5013.646} C_VEL
LIN {X 0,Y 517.705,Z 667.394,A -85,B 0,C 180,E1 -5014.684,E2 -5014.684} C_VEL
LIN {X 0,Y 517.354,Z 677.09,A -85,B 0,C 180,E1 -5015.781,E2 -5015.781} C_VEL
LIN {X 0,Y 517.049,Z 685.989,A -85,B 0,C 180,E1 -5016.997,E2 -5016.997} C_VEL
LIN {X 0,Y 516.822,Z 694.64,A -85,B 0,C 180,E1 -5018.46,E2 -5018.46} C_VEL
LIN {X 0,Y 516.608,Z 701.072,A -85,B 0,C 180,E1 -5019.83,E2 -5019.83} C_VEL
LIN {X 0,Y 516.502,Z 705.321,A -85,B 0,C 180,E1 -5020.94,E2 -5020.94} C_VEL
LIN {X 0,Y 516.441,Z 709.362,A -85,B 0,C 180,E1 -5022.286,E2 -5022.286} C_VEL
LIN {X 0,Y 516.317,Z 711.914,A -85,B 0,C 180,E1 -5023.391,E2 -5023.391} C_VEL
LIN {X 0,Y 516.288,Z 713.378,A -85,B 0,C 180,E1 -5024.202,E2 -5024.202} C_VEL
LIN {X 0,Y 516.305,Z 715.098,A -85,B 0,C 180,E1 -5025.817,E2 -5025.817} C_VEL
LIN {X 0,Y 516.284,Z 715.475,A -85,B 0,C 180,E1 -5026.62,E2 -5026.62} C_VEL
LIN {X 0,Y 516.321,Z 715.179,A -85,B 0,C 180,E1 -5028.219,E2 -5028.219} C_VEL
LIN {X 0,Y 516.316,Z 713.512,A -85,B 0,C 180,E1 -5029.808,E2 -5029.808} C_VEL
LIN {X 0,Y 516.321,Z 712.242,A -85,B 0,C 180,E1 -5030.6,E2 -5030.6} C_VEL
LIN {X 0,Y 516.443,Z 708.485,A -85,B 0,C 180,E1 -5032.179,E2 -5032.179} C_VEL
LIN {X 0,Y 516.582,Z 705.016,A -85,B 0,C 180,E1 -5033.284,E2 -5033.284} C_VEL
LIN {X 0,Y 516.643,Z 700.091,A -85,B 0,C 180,E1 -5034.536,E2 -5034.536} C_VEL
LIN {X 0,Y 516.86,Z 693.337,A -85,B 0,C 180,E1 -5035.907,E2 -5035.907} C_VEL
LIN {X 0,Y 517.05,Z 686.314,A -85,B 0,C 180,E1 -5037.079,E2 -5037.079} C_VEL
LIN {X 0,Y 517.383,Z 677.858,A -85,B 0,C 180,E1 -5038.249,E2 -5038.249} C_VEL
LIN {X 0,Y 517.691,Z 667.651,A -85,B 0,C 180,E1 -5039.417,E2 -5039.417} C_VEL
LIN {X 0,Y 518.107,Z 657.242,A -85,B 0,C 180,E1 -5040.389,E2 -5040.389} C_VEL
LIN {X 0,Y 518.494,Z 645.875,A -85,B 0,C 180,E1 -5041.262,E2 -5041.262} C_VEL
LIN {X 0,Y 518.851,Z 633.352,A -85,B 0,C 180,E1 -5042.038,E2 -5042.038} C_VEL
LIN {X 0,Y 519.13,Z 619.112,A -85,B 0,C 180,E1 -5042.716,E2 -5042.716} C_VEL
LIN {X 0,Y 519.307,Z 605.177,A -85,B 0,C 180,E1 -5043.201,E2 -5043.201} C_VEL
LIN {X 0,Y 519.425,Z 591.559,A -85,B 0,C 180,E1 -5043.515,E2 -5043.515} C_VEL
LIN {X 0,Y 519.541,Z 544.207,A -85,B 0,C 180,E1 -5044.185,E2 -5044.185} C_VEL
LIN {X 0,Y 516.948,Z 536.091,A -85,B 0,C 180,E1 -5044.386,E2 -5044.386} C_VEL
LIN {X 0,Y 516.998,Z 536.086,A -85,B 0,C 180,E1 -5047.096,E2 -5047.096} C_VEL
LIN {X 0,Y 516.95,Z 536.094,A -85,B 0,C 180,E1 -5049.39,E2 -5049.39} C_VEL
LIN {X 0,Y 516.98,Z 536.091,A -85,B 0,C 180,E1 -5051.824,E2 -5051.824} C_VEL
LIN {X 0,Y 516.941,Z 536.094,A -85,B 0,C 180,E1 -5055.147,E2 -5055.147} C_VEL
LIN {X 0,Y 516.922,Z 536.093,A -85,B 0,C 180,E1 -5058.223,E2 -5058.223} C_VEL
LIN {X 0,Y 516.91,Z 536.093,A -85,B 0,C 180,E1 -5060.702,E2 -5060.702} C_VEL
LIN {X 0,Y 516.909,Z 536.094,A -85,B 0,C 180,E1 -5064.072,E2 -5064.072} C_VEL
LIN {X 0,Y 516.927,Z 536.09,A -85,B 0,C 180,E1 -5066.658,E2 -5066.658} C_VEL
LIN {X 0,Y 516.918,Z 536.095,A -85,B 0,C 180,E1 -5069.526,E2 -5069.526} C_VEL
LIN {X 0,Y 516.899,Z 536.09,A -85,B 0,C 180,E1 -5072.545,E2 -5072.545} C_VEL
LIN {X 0,Y 516.871,Z 536.102,A -85,B 0,C 180,E1 -5075.331,E2 -5075.331} C_VEL
LIN {X 0,Y 516.88,Z 536.096,A -85,B 0,C 180,E1 -5077.944,E2 -5077.944} C_VEL
LIN {X 0,Y 516.885,Z 536.097,A -85,B 0,C 180,E1 -5080.742,E2 -5080.742} C_VEL
LIN {X 0,Y 516.904,Z 536.095,A -85,B 0,C 180,E1 -5082.83,E2 -5082.83} C_VEL
LIN {X 0,Y 516.922,Z 536.096,A -85,B 0,C 180,E1 -5085.011,E2 -5085.011} C_VEL
LIN {X 0,Y 516.914,Z 536.091,A -85,B 0,C 180,E1 -5088.399,E2 -5088.399} C_VEL
LIN {X 0,Y 516.883,Z 536.104,A -85,B 0,C 180,E1 -5091.285,E2 -5091.285} C_VEL
LIN {X 0,Y 516.888,Z 536.098,A -85,B 0,C 180,E1 -5094.222,E2 -5094.222} C_VEL
LIN {X 0,Y 516.94,Z 536.235,A -85,B 0,C 180,E1 -5097.084,E2 -5097.084} C_VEL
LIN {X 0,Y 519.605,Z 548.71,A -85,B 0,C 180,E1 -5099.298,E2 -5099.298} C_VEL
LIN {X 0,Y 519.317,Z 561.102,A -85,B 0,C 180,E1 -5101.282,E2 -5101.282} C_VEL
LIN {X 0,Y 518.823,Z 579.061,A -85,B 0,C 180,E1 -5104.097,E2 -5104.097} C_VEL
LIN {X 0,Y 518.379,Z 597.038,A -85,B 0,C 180,E1 -5106.849,E2 -5106.849} C_VEL
LIN {X 0,Y 517.953,Z 616.47,A -85,B 0,C 180,E1 -5109.768,E2 -5109.768} C_VEL
LIN {X 0,Y 517.572,Z 636.042,A -85,B 0,C 180,E1 -5112.619,E2 -5112.619} C_VEL
LIN {X 0,Y 517.313,Z 649.379,A -85,B 0,C 180,E1 -5114.571,E2 -5114.571} C_VEL
LIN {X 0,Y 519.14,Z 663.242,A -85,B 0,C 180,E1 -5114.834,E2 -5114.834} C_VEL
LIN {X 0,Y 518.701,Z 753.354,A -85,B 0,C 180,E1 -5116.11,E2 -5116.11} C_VEL
LIN {X 0,Y 518.475,Z 767.203,A -85,B 0,C 180,E1 -5116.403,E2 -5116.403} C_VEL
LIN {X 0,Y 518.26,Z 779.658,A -85,B 0,C 180,E1 -5116.822,E2 -5116.822} C_VEL
LIN {X 0,Y 517.964,Z 791.374,A -85,B 0,C 180,E1 -5117.362,E2 -5117.362} C_VEL
LIN {X 0,Y 517.722,Z 802.985,A -85,B 0,C 180,E1 -5118.061,E2 -5118.061} C_VEL
LIN {X 0,Y 517.38,Z 814.576,A -85,B 0,C 180,E1 -5118.938,E2 -5118.938} C_VEL
LIN {X 0,Y 517.066,Z 824.037,A -85,B 0,C 180,E1 -5119.823,E2 -5119.823} C_VEL
LIN {X 0,Y 516.844,Z 832.689,A -85,B 0,C 180,E1 -5120.807,E2 -5120.807} C_VEL
LIN {X 0,Y 516.641,Z 841.125,A -85,B 0,C 180,E1 -5121.985,E2 -5121.985} C_VEL
LIN {X 0,Y 516.479,Z 848.066,A -85,B 0,C 180,E1 -5123.202,E2 -5123.202} C_VEL
LIN {X 0,Y 516.405,Z 853.949,A -85,B 0,C 180,E1 -5124.534,E2 -5124.534} C_VEL
LIN {X 0,Y 516.344,Z 857.894,A -85,B 0,C 180,E1 -5125.707,E2 -5125.707} C_VEL
LIN {X 0,Y 516.283,Z 860.811,A -85,B 0,C 180,E1 -5126.879,E2 -5126.879} C_VEL
LIN {X 0,Y 516.26,Z 862.198,A -85,B 0,C 180,E1 -5127.66,E2 -5127.66} C_VEL
LIN {X 0,Y 516.16,Z 863.786,A -85,B 0,C 180,E1 -5129.22,E2 -5129.22} C_VEL
LIN {X 0,Y 516.154,Z 864,A -85,B 0,C 180,E1 -5130,E2 -5130} C_VEL
LIN {X 0,Y 516.192,Z 863.181,A -85,B 0,C 180,E1 -5131.561,E2 -5131.561} C_VEL
LIN {X 0,Y 516.26,Z 862.193,A -85,B 0,C 180,E1 -5132.341,E2 -5132.341} C_VEL
LIN {X 0,Y 516.283,Z 860.807,A -85,B 0,C 180,E1 -5133.122,E2 -5133.122} C_VEL
LIN {X 0,Y 516.344,Z 857.895,A -85,B 0,C 180,E1 -5134.294,E2 -5134.294} C_VEL
LIN {X 0,Y 516.405,Z 853.948,A -85,B 0,C 180,E1 -5135.467,E2 -5135.467} C_VEL
LIN {X 0,Y 516.487,Z 848.01,A -85,B 0,C 180,E1 -5136.808,E2 -5136.808} C_VEL
LIN {X 0,Y 516.641,Z 841.118,A -85,B 0,C 180,E1 -5138.015,E2 -5138.015} C_VEL
LIN {X 0,Y 516.845,Z 832.664,A -85,B 0,C 180,E1 -5139.194,E2 -5139.194} C_VEL
LIN {X 0,Y 517.067,Z 823.925,A -85,B 0,C 180,E1 -5140.178,E2 -5140.178} C_VEL
LIN {X 0,Y 517.399,Z 813.161,A -85,B 0,C 180,E1 -5141.161,E2 -5141.161} C_VEL
LIN {X 0,Y 517.651,Z 802.335,A -85,B 0,C 180,E1 -5141.961,E2 -5141.961} C_VEL
LIN {X 0,Y 517.973,Z 790.823,A -85,B 0,C 180,E1 -5142.638,E2 -5142.638} C_VEL
LIN {X 0,Y 518.206,Z 778.835,A -85,B 0,C 180,E1 -5143.181,E2 -5143.181} C_VEL
LIN {X 0,Y 518.457,Z 765.094,A -85,B 0,C 180,E1 -5143.623,E2 -5143.623} C_VEL
LIN {X 0,Y 518.67,Z 751.504,A -85,B 0,C 180,E1 -5143.892,E2 -5143.892} C_VEL
LIN {X 0,Y 518.952,Z 660.818,A -85,B 0,C 180,E1 -5145.171,E2 -5145.171} C_VEL
LIN {X 0,Y 517.372,Z 650.157,A -85,B 0,C 180,E1 -5145.367,E2 -5145.367} C_VEL
LIN {X 0,Y 517.281,Z 647.749,A -85,B 0,C 180,E1 -5145.415,E2 -5145.415} C_VEL
LIN {X 0,Y 517.647,Z 625.957,A -85,B 0,C 180,E1 -5148.401,E2 -5148.401} C_VEL
LIN {X 0,Y 517.828,Z 604.803,A -85,B 0,C 180,E1 -5151.288,E2 -5151.288} C_VEL
LIN {X 0,Y 517.999,Z 584.999,A -85,B 0,C 180,E1 -5154.019,E2 -5154.019} C_VEL
LIN {X 0,Y 518.058,Z 563.374,A -85,B 0,C 180,E1 -5157.031,E2 -5157.031} C_VEL
LIN {X 0,Y 518.061,Z 543.234,A -85,B 0,C 180,E1 -5159.903,E2 -5159.903} C_VEL
LIN {X 0,Y 516.987,Z 536.091,A -85,B 0,C 180,E1 -5160.972,E2 -5160.972} C_VEL
LIN {X 0,Y 516.916,Z 536.093,A -85,B 0,C 180,E1 -5163.967,E2 -5163.967} C_VEL
LIN {X 0,Y 516.881,Z 536.102,A -85,B 0,C 180,E1 -5166.746,E2 -5166.746} C_VEL
LIN {X 0,Y 516.887,Z 536.095,A -85,B 0,C 180,E1 -5169.721,E2 -5169.721} C_VEL
LIN {X 0,Y 516.916,Z 536.091,A -85,B 0,C 180,E1 -5171.775,E2 -5171.775} C_VEL
LIN {X 0,Y 516.928,Z 536.096,A -85,B 0,C 180,E1 -5175.01,E2 -5175.01} C_VEL
LIN {X 0,Y 516.922,Z 536.095,A -85,B 0,C 180,E1 -5178.398,E2 -5178.398} C_VEL
LIN {X 0,Y 516.887,Z 536.097,A -85,B 0,C 180,E1 -5181.284,E2 -5181.284} C_VEL
LIN {X 0,Y 516.875,Z 536.1,A -85,B 0,C 180,E1 -5184.22,E2 -5184.22} C_VEL
LIN {X 0,Y 516.899,Z 536.097,A -85,B 0,C 180,E1 -5187.053,E2 -5187.053} C_VEL
LIN {X 0,Y 516.897,Z 536.095,A -85,B 0,C 180,E1 -5189.796,E2 -5189.796} C_VEL
LIN {X 0,Y 516.933,Z 536.098,A -85,B 0,C 180,E1 -5192.467,E2 -5192.467} C_VEL
LIN {X 0,Y 516.916,Z 536.095,A -85,B 0,C 180,E1 -5195.072,E2 -5195.072} C_VEL
LIN {X 0,Y 516.891,Z 536.103,A -85,B 0,C 180,E1 -5198.462,E2 -5198.462} C_VEL
LIN {X 0,Y 516.905,Z 536.097,A -85,B 0,C 180,E1 -5200.955,E2 -5200.955} C_VEL
LIN {X 0,Y 516.912,Z 536.097,A -85,B 0,C 180,E1 -5203.512,E2 -5203.512} C_VEL
LIN {X 0,Y 520.033,Z 545.513,A -85,B 0,C 180,E1 -5203.74,E2 -5203.74} C_VEL
LIN {X 0,Y 520.017,Z 578.87,A -85,B 0,C 180,E1 -5204.223,E2 -5204.223} C_VEL
LIN {X 0,Y 519.911,Z 593.649,A -85,B 0,C 180,E1 -5204.591,E2 -5204.591} C_VEL
LIN {X 0,Y 519.76,Z 608.178,A -85,B 0,C 180,E1 -5205.113,E2 -5205.113} C_VEL
LIN {X 0,Y 519.447,Z 622.644,A -85,B 0,C 180,E1 -5205.804,E2 -5205.804} C_VEL
LIN {X 0,Y 519.122,Z 635.687,A -85,B 0,C 180,E1 -5206.594,E2 -5206.594} C_VEL
LIN {X 0,Y 518.819,Z 647.662,A -85,B 0,C 180,E1 -5207.482,E2 -5207.482} C_VEL
LIN {X 0,Y 518.426,Z 658.686,A -85,B 0,C 180,E1 -5208.465,E2 -5208.465} C_VEL
LIN {X 0,Y 517.957,Z 669.753,A -85,B 0,C 180,E1 -5209.642,E2 -5209.642} C_VEL
LIN {X 0,Y 517.643,Z 680.409,A -85,B 0,C 180,E1 -5211.017,E2 -5211.017} C_VEL
LIN {X 0,Y 517.293,Z 689.567,A -85,B 0,C 180,E1 -5212.456,E2 -5212.456} C_VEL
LIN {X 0,Y 517.046,Z 696.392,A -85,B 0,C 180,E1 -5213.757,E2 -5213.757} C_VEL
LIN {X 0,Y 516.819,Z 703.109,A -85,B 0,C 180,E1 -5215.32,E2 -5215.32} C_VEL
LIN {X 0,Y 516.664,Z 708.352,A -85,B 0,C 180,E1 -5216.881,E2 -5216.881} C_VEL
LIN {X 0,Y 516.508,Z 712.29,A -85,B 0,C 180,E1 -5218.44,E2 -5218.44} C_VEL
LIN {X 0,Y 516.437,Z 715.018,A -85,B 0,C 180,E1 -5220,E2 -5220} C_VEL
LIN {X 0,Y 516.41,Z 716.614,A -85,B 0,C 180,E1 -5221.559,E2 -5221.559} C_VEL
LIN {X 0,Y 516.459,Z 717.088,A -85,B 0,C 180,E1 -5223.12,E2 -5223.12} C_VEL
LIN {X 0,Y 516.456,Z 716.45,A -85,B 0,C 180,E1 -5224.683,E2 -5224.683} C_VEL
LIN {X 0,Y 516.522,Z 714.665,A -85,B 0,C 180,E1 -5226.249,E2 -5226.249} C_VEL
LIN {X 0,Y 516.528,Z 711.727,A -85,B 0,C 180,E1 -5227.82,E2 -5227.82} C_VEL
LIN {X 0,Y 516.64,Z 707.55,A -85,B 0,C 180,E1 -5229.395,E2 -5229.395} C_VEL
LIN {X 0,Y 516.782,Z 702.013,A -85,B 0,C 180,E1 -5230.975,E2 -5230.975} C_VEL
LIN {X 0,Y 517.018,Z 694.937,A -85,B 0,C 180,E1 -5232.561,E2 -5232.561} C_VEL
LIN {X 0,Y 517.281,Z 687.303,A -85,B 0,C 180,E1 -5233.955,E2 -5233.955} C_VEL
LIN {X 0,Y 517.617,Z 678.737,A -85,B 0,C 180,E1 -5235.257,E2 -5235.257} C_VEL
LIN {X 0,Y 518.014,Z 668.528,A -85,B 0,C 180,E1 -5236.553,E2 -5236.553} C_VEL
LIN {X 0,Y 518.422,Z 657.123,A -85,B 0,C 180,E1 -5237.759,E2 -5237.759} C_VEL
LIN {X 0,Y 518.856,Z 645.24,A -85,B 0,C 180,E1 -5238.805,E2 -5238.805} C_VEL
LIN {X 0,Y 519.27,Z 633.411,A -85,B 0,C 180,E1 -5239.674,E2 -5239.674} C_VEL
LIN {X 0,Y 519.666,Z 619.929,A -85,B 0,C 180,E1 -5240.483,E2 -5240.483} C_VEL
LIN {X 0,Y 520.014,Z 605.516,A -85,B 0,C 180,E1 -5241.166,E2 -5241.166} C_VEL
LIN {X 0,Y 520.244,Z 590.437,A -85,B 0,C 180,E1 -5241.703,E2 -5241.703} C_VEL
LIN {X 0,Y 520.415,Z 574.648,A -85,B 0,C 180,E1 -5242.087,E2 -5242.087} C_VEL
LIN {X 0,Y 520.419,Z 545.963,A -85,B 0,C 180,E1 -5242.52,E2 -5242.52} C_VEL
LIN {X 0,Y 516.864,Z 536.101,A -85,B 0,C 180,E1 -5242.8,E2 -5242.8} C_VEL
LIN {X 0,Y 516.931,Z 536.097,A -85,B 0,C 180,E1 -5245.789,E2 -5245.789} C_VEL
LIN {X 0,Y 516.921,Z 536.094,A -85,B 0,C 180,E1 -5248.415,E2 -5248.415} C_VEL
LIN {X 0,Y 516.89,Z 536.093,A -85,B 0,C 180,E1 -5251.109,E2 -5251.109} C_VEL
LIN {X 0,Y 516.909,Z 536.098,A -85,B 0,C 180,E1 -5253.966,E2 -5253.966} C_VEL
LIN {X 0,Y 516.877,Z 536.096,A -85,B 0,C 180,E1 -5256.746,E2 -5256.746} C_VEL
LIN {X 0,Y 516.884,Z 536.096,A -85,B 0,C 180,E1 -5259.721,E2 -5259.721} C_VEL
LIN {X 0,Y 516.884,Z 536.095,A -85,B 0,C 180,E1 -5260.865,E2 -5260.865} C_VEL
LIN {X 0,Y 516.215,Z 536.178,A -85,B 0,C 180,E1 -5261.516,E2 -5261.516} C_VEL
LIN {X 0,Y 513.349,Z 536.541,A -85,B 0,C 180,E1 -5262.572,E2 -5262.572} C_VEL
LIN {X 0,Y 510.932,Z 536.846,A -85,B 0,C 180,E1 -5263.423,E2 -5263.423} C_VEL
LIN {X 0,Y 509.903,Z 536.973,A -85,B 0,C 180,E1 -5264.08,E2 -5264.08} C_VEL
LIN {X 0,Y 509.824,Z 536.98,A -85,B 0,C 180,E1 -5264.303,E2 -5264.303} C_VEL
LIN {X 0,Y 509.834,Z 536.972,A -85,B 0,C 180,E1 -5267.51,E2 -5267.51} C_VEL
LIN {X 0,Y 509.847,Z 536.976,A -85,B 0,C 180,E1 -5270.647,E2 -5270.647} C_VEL
LIN {X 0,Y 509.827,Z 536.973,A -85,B 0,C 180,E1 -5273.647,E2 -5273.647} C_VEL
LIN {X 0,Y 509.861,Z 536.979,A -85,B 0,C 180,E1 -5276.539,E2 -5276.539} C_VEL
LIN {X 0,Y 509.845,Z 536.971,A -85,B 0,C 180,E1 -5279.334,E2 -5279.334} C_VEL
LIN {X 0,Y 509.893,Z 536.966,A -85,B 0,C 180,E1 -5282.054,E2 -5282.054} C_VEL
LIN {X 0,Y 509.877,Z 536.976,A -85,B 0,C 180,E1 -5284.704,E2 -5284.704} C_VEL
LIN {X 0,Y 509.836,Z 536.973,A -85,B 0,C 180,E1 -5287.455,E2 -5287.455} C_VEL
LIN {X 0,Y 509.916,Z 536.962,A -85,B 0,C 180,E1 -5289.844,E2 -5289.844} C_VEL
LIN {X 0,Y 509.884,Z 536.97,A -85,B 0,C 180,E1 -5293.174,E2 -5293.174} C_VEL
LIN {X 0,Y 509.863,Z 536.969,A -85,B 0,C 180,E1 -5295.634,E2 -5295.634} C_VEL
LIN {X 0,Y 509.901,Z 536.964,A -85,B 0,C 180,E1 -5298.123,E2 -5298.123} C_VEL
LIN {X 0,Y 509.915,Z 536.967,A -85,B 0,C 180,E1 -5301.279,E2 -5301.279} C_VEL
LIN {X 0,Y 509.977,Z 536.955,A -85,B 0,C 180,E1 -5303.67,E2 -5303.67} C_VEL
LIN {X 0,Y 510.054,Z 536.947,A -85,B 0,C 180,E1 -5307.63,E2 -5307.63} C_VEL
LIN {X 0,Y 510.062,Z 536.948,A -85,B 0,C 180,E1 -5310.789,E2 -5310.789} C_VEL
LIN {X 0,Y 509.956,Z 536.966,A -85,B 0,C 180,E1 -5313.16,E2 -5313.16} C_VEL
LIN {X 0,Y 509.952,Z 536.957,A -85,B 0,C 180,E1 -5316.329,E2 -5316.329} C_VEL
LIN {X 0,Y 509.913,Z 536.964,A -85,B 0,C 180,E1 -5318.72,E2 -5318.72} C_VEL
LIN {X 0,Y 509.949,Z 536.96,A -85,B 0,C 180,E1 -5321.93,E2 -5321.93} C_VEL
LIN {X 0,Y 509.89,Z 536.972,A -85,B 0,C 180,E1 -5325.241,E2 -5325.241} C_VEL
LIN {X 0,Y 509.886,Z 536.968,A -85,B 0,C 180,E1 -5328.001,E2 -5328.001} C_VEL
LIN {X 0,Y 509.847,Z 536.973,A -85,B 0,C 180,E1 -5331.001,E2 -5331.001} C_VEL
LIN {X 0,Y 509.833,Z 536.982,A -85,B 0,C 180,E1 -5333.563,E2 -5333.563} C_VEL
LIN {X 0,Y 509.91,Z 536.963,A -85,B 0,C 180,E1 -5336.379,E2 -5336.379} C_VEL
LIN {X 0,Y 509.882,Z 536.966,A -85,B 0,C 180,E1 -5338.843,E2 -5338.843} C_VEL
LIN {X 0,Y 509.823,Z 536.981,A -85,B 0,C 180,E1 -5341.589,E2 -5341.589} C_VEL
LIN {X 0,Y 509.85,Z 536.971,A -85,B 0,C 180,E1 -5344.413,E2 -5344.413} C_VEL
LIN {X 0,Y 509.815,Z 536.977,A -85,B 0,C 180,E1 -5347.34,E2 -5347.34} C_VEL
LIN {X 0,Y 509.856,Z 536.972,A -85,B 0,C 180,E1 -5350.38,E2 -5350.38} C_VEL
LIN {X 0,Y 509.819,Z 536.974,A -85,B 0,C 180,E1 -5353.062,E2 -5353.062} C_VEL
LIN {X 0,Y 509.826,Z 536.98,A -85,B 0,C 180,E1 -5355.792,E2 -5355.792} C_VEL
LIN {X 0,Y 509.862,Z 536.971,A -85,B 0,C 180,E1 -5358.576,E2 -5358.576} C_VEL
LIN {X 0,Y 509.851,Z 536.975,A -85,B 0,C 180,E1 -5361.785,E2 -5361.785} C_VEL
LIN {X 0,Y 509.842,Z 536.974,A -85,B 0,C 180,E1 -5364.623,E2 -5364.623} C_VEL
LIN {X 0,Y 509.861,Z 536.971,A -85,B 0,C 180,E1 -5367.481,E2 -5367.481} C_VEL
LIN {X 0,Y 509.885,Z 536.971,A -85,B 0,C 180,E1 -5369.422,E2 -5369.422} C_VEL
LIN {X 0,Y 512.993,Z 546.045,A -85,B 0,C 180,E1 -5369.665,E2 -5369.665} C_VEL
LIN {X 0,Y 512.685,Z 594.486,A -85,B 0,C 180,E1 -5370.387,E2 -5370.387} C_VEL
LIN {X 0,Y 512.482,Z 608.66,A -85,B 0,C 180,E1 -5370.755,E2 -5370.755} C_VEL
LIN {X 0,Y 512.288,Z 621.695,A -85,B 0,C 180,E1 -5371.249,E2 -5371.249} C_VEL
LIN {X 0,Y 511.995,Z 634.231,A -85,B 0,C 180,E1 -5371.874,E2 -5371.874} C_VEL
LIN {X 0,Y 511.596,Z 645.829,A -85,B 0,C 180,E1 -5372.6,E2 -5372.6} C_VEL
LIN {X 0,Y 511.221,Z 658.358,A -85,B 0,C 180,E1 -5373.582,E2 -5373.582} C_VEL
LIN {X 0,Y 510.817,Z 668.358,A -85,B 0,C 180,E1 -5374.536,E2 -5374.536} C_VEL
LIN {X 0,Y 510.44,Z 677.714,A -85,B 0,C 180,E1 -5375.604,E2 -5375.604} C_VEL
LIN {X 0,Y 510.099,Z 686.954,A -85,B 0,C 180,E1 -5376.88,E2 -5376.88} C_VEL
LIN {X 0,Y 509.845,Z 695.63,A -85,B 0,C 180,E1 -5378.363,E2 -5378.363} C_VEL
LIN {X 0,Y 509.625,Z 702.415,A -85,B 0,C 180,E1 -5379.833,E2 -5379.833} C_VEL
LIN {X 0,Y 509.484,Z 707.023,A -85,B 0,C 180,E1 -5381.085,E2 -5381.085} C_VEL
LIN {X 0,Y 509.436,Z 710.615,A -85,B 0,C 180,E1 -5382.332,E2 -5382.332} C_VEL
LIN {X 0,Y 509.318,Z 712.554,A -85,B 0,C 180,E1 -5383.156,E2 -5383.156} C_VEL
LIN {X 0,Y 509.277,Z 715.175,A -85,B 0,C 180,E1 -5384.8,E2 -5384.8} C_VEL
LIN {X 0,Y 509.264,Z 716.424,A -85,B 0,C 180,E1 -5386.432,E2 -5386.432} C_VEL
LIN {X 0,Y 509.293,Z 716.285,A -85,B 0,C 180,E1 -5388.054,E2 -5388.054} C_VEL
LIN {X 0,Y 509.298,Z 714.803,A -85,B 0,C 180,E1 -5389.666,E2 -5389.666} C_VEL
LIN {X 0,Y 509.356,Z 711.947,A -85,B 0,C 180,E1 -5391.271,E2 -5391.271} C_VEL
LIN {X 0,Y 509.502,Z 708.856,A -85,B 0,C 180,E1 -5392.471,E2 -5392.471} C_VEL
LIN {X 0,Y 509.607,Z 704.949,A -85,B 0,C 180,E1 -5393.666,E2 -5393.666} C_VEL
LIN {X 0,Y 509.717,Z 700.109,A -85,B 0,C 180,E1 -5394.858,E2 -5394.858} C_VEL
LIN {X 0,Y 509.966,Z 693.14,A -85,B 0,C 180,E1 -5396.247,E2 -5396.247} C_VEL
LIN {X 0,Y 510.216,Z 684.468,A -85,B 0,C 180,E1 -5397.632,E2 -5397.632} C_VEL
LIN {X 0,Y 510.637,Z 675.347,A -85,B 0,C 180,E1 -5398.817,E2 -5398.817} C_VEL
LIN {X 0,Y 510.931,Z 665.303,A -85,B 0,C 180,E1 -5399.902,E2 -5399.902} C_VEL
LIN {X 0,Y 511.374,Z 654.178,A -85,B 0,C 180,E1 -5400.886,E2 -5400.886} C_VEL
LIN {X 0,Y 511.807,Z 641.845,A -85,B 0,C 180,E1 -5401.771,E2 -5401.771} C_VEL
LIN {X 0,Y 512.136,Z 628.768,A -85,B 0,C 180,E1 -5402.507,E2 -5402.507} C_VEL
LIN {X 0,Y 512.38,Z 615.002,A -85,B 0,C 180,E1 -5403.096,E2 -5403.096} C_VEL
LIN {X 0,Y 512.55,Z 601.328,A -85,B 0,C 180,E1 -5403.513,E2 -5403.513} C_VEL
LIN {X 0,Y 512.626,Z 587.32,A -85,B 0,C 180,E1 -5403.783,E2 -5403.783} C_VEL
LIN {X 0,Y 512.744,Z 545.758,A -85,B 0,C 180,E1 -5404.371,E2 -5404.371} C_VEL
LIN {X 0,Y 509.889,Z 536.97,A -85,B 0,C 180,E1 -5404.596,E2 -5404.596} C_VEL
LIN {X 0,Y 509.97,Z 536.962,A -85,B 0,C 180,E1 -5407.145,E2 -5407.145} C_VEL
LIN {X 0,Y 509.861,Z 536.973,A -85,B 0,C 180,E1 -5410.323,E2 -5410.323} C_VEL
LIN {X 0,Y 509.877,Z 536.971,A -85,B 0,C 180,E1 -5412.741,E2 -5412.741} C_VEL
LIN {X 0,Y 509.89,Z 536.974,A -85,B 0,C 180,E1 -5415.242,E2 -5415.242} C_VEL
LIN {X 0,Y 509.886,Z 536.971,A -85,B 0,C 180,E1 -5418.001,E2 -5418.001} C_VEL
LIN {X 0,Y 509.848,Z 536.975,A -85,B 0,C 180,E1 -5421.002,E2 -5421.002} C_VEL
LIN {X 0,Y 509.834,Z 536.98,A -85,B 0,C 180,E1 -5423.564,E2 -5423.564} C_VEL
LIN {X 0,Y 509.912,Z 536.963,A -85,B 0,C 180,E1 -5426.38,E2 -5426.38} C_VEL
LIN {X 0,Y 509.879,Z 536.968,A -85,B 0,C 180,E1 -5428.844,E2 -5428.844} C_VEL
LIN {X 0,Y 509.825,Z 536.976,A -85,B 0,C 180,E1 -5431.59,E2 -5431.59} C_VEL
LIN {X 0,Y 509.849,Z 536.969,A -85,B 0,C 180,E1 -5434.414,E2 -5434.414} C_VEL
LIN {X 0,Y 509.816,Z 536.981,A -85,B 0,C 180,E1 -5437.341,E2 -5437.341} C_VEL
LIN {X 0,Y 509.837,Z 536.973,A -85,B 0,C 180,E1 -5440.383,E2 -5440.383} C_VEL
LIN {X 0,Y 509.839,Z 536.979,A -85,B 0,C 180,E1 -5443.065,E2 -5443.065} C_VEL
LIN {X 0,Y 509.83,Z 536.975,A -85,B 0,C 180,E1 -5445.793,E2 -5445.793} C_VEL
LIN {X 0,Y 509.856,Z 536.972,A -85,B 0,C 180,E1 -5448.575,E2 -5448.575} C_VEL
LIN {X 0,Y 509.851,Z 536.974,A -85,B 0,C 180,E1 -5451.787,E2 -5451.787} C_VEL
LIN {X 0,Y 509.844,Z 536.978,A -85,B 0,C 180,E1 -5454.624,E2 -5454.624} C_VEL
LIN {X 0,Y 509.878,Z 537.105,A -85,B 0,C 180,E1 -5456.834,E2 -5456.834} C_VEL
LIN {X 0,Y 512.59,Z 549.426,A -85,B 0,C 180,E1 -5459.06,E2 -5459.06} C_VEL
LIN {X 0,Y 512.629,Z 556.461,A -85,B 0,C 180,E1 -5460.225,E2 -5460.225} C_VEL
LIN {X 0,Y 512.022,Z 574.699,A -85,B 0,C 180,E1 -5463.15,E2 -5463.15} C_VEL
LIN {X 0,Y 511.465,Z 594.876,A -85,B 0,C 180,E1 -5466.302,E2 -5466.302} C_VEL
LIN {X 0,Y 511.006,Z 614.25,A -85,B 0,C 180,E1 -5469.265,E2 -5469.265} C_VEL
LIN {X 0,Y 510.557,Z 635.054,A -85,B 0,C 180,E1 -5472.372,E2 -5472.372} C_VEL
LIN {X 0,Y 510.271,Z 648.194,A -85,B 0,C 180,E1 -5474.311,E2 -5474.311} C_VEL
LIN {X 0,Y 512.301,Z 663.421,A -85,B 0,C 180,E1 -5474.62,E2 -5474.62} C_VEL
LIN {X 0,Y 511.874,Z 745.023,A -85,B 0,C 180,E1 -5475.794,E2 -5475.794} C_VEL
LIN {X 0,Y 511.658,Z 762.698,A -85,B 0,C 180,E1 -5476.117,E2 -5476.117} C_VEL
LIN {X 0,Y 511.343,Z 776.132,A -85,B 0,C 180,E1 -5476.539,E2 -5476.539} C_VEL
LIN {X 0,Y 511.041,Z 788.472,A -85,B 0,C 180,E1 -5477.087,E2 -5477.087} C_VEL
LIN {X 0,Y 510.741,Z 800.048,A -85,B 0,C 180,E1 -5477.761,E2 -5477.761} C_VEL
LIN {X 0,Y 510.374,Z 811.175,A -85,B 0,C 180,E1 -5478.584,E2 -5478.584} C_VEL
LIN {X 0,Y 510.075,Z 821.047,A -85,B 0,C 180,E1 -5479.481,E2 -5479.481} C_VEL
LIN {X 0,Y 509.815,Z 830.067,A -85,B 0,C 180,E1 -5480.479,E2 -5480.479} C_VEL
LIN {X 0,Y 509.612,Z 838.887,A -85,B 0,C 180,E1 -5481.675,E2 -5481.675} C_VEL
LIN {X 0,Y 509.419,Z 845.941,A -85,B 0,C 180,E1 -5482.868,E2 -5482.868} C_VEL
LIN {X 0,Y 509.368,Z 851.608,A -85,B 0,C 180,E1 -5484.061,E2 -5484.061} C_VEL
LIN {X 0,Y 509.19,Z 856.036,A -85,B 0,C 180,E1 -5485.25,E2 -5485.25} C_VEL
LIN {X 0,Y 509.286,Z 858.41,A -85,B 0,C 180,E1 -5486.044,E2 -5486.044} C_VEL
LIN {X 0,Y 509.201,Z 860.313,A -85,B 0,C 180,E1 -5486.836,E2 -5486.836} C_VEL
LIN {X 0,Y 509.189,Z 861.746,A -85,B 0,C 180,E1 -5487.627,E2 -5487.627} C_VEL
LIN {X 0,Y 509.073,Z 863.373,A -85,B 0,C 180,E1 -5489.209,E2 -5489.209} C_VEL
LIN {X 0,Y 509.066,Z 863.591,A -85,B 0,C 180,E1 -5490,E2 -5490} C_VEL
LIN {X 0,Y 509.073,Z 863.367,A -85,B 0,C 180,E1 -5490.791,E2 -5490.791} C_VEL
LIN {X 0,Y 509.189,Z 861.73,A -85,B 0,C 180,E1 -5492.374,E2 -5492.374} C_VEL
LIN {X 0,Y 509.201,Z 860.285,A -85,B 0,C 180,E1 -5493.165,E2 -5493.165} C_VEL
LIN {X 0,Y 509.252,Z 857.263,A -85,B 0,C 180,E1 -5494.354,E2 -5494.354} C_VEL
LIN {X 0,Y 509.344,Z 853.165,A -85,B 0,C 180,E1 -5495.543,E2 -5495.543} C_VEL
LIN {X 0,Y 509.417,Z 847.195,A -85,B 0,C 180,E1 -5496.865,E2 -5496.865} C_VEL
LIN {X 0,Y 509.573,Z 839.933,A -85,B 0,C 180,E1 -5498.127,E2 -5498.127} C_VEL
LIN {X 0,Y 509.783,Z 831.359,A -85,B 0,C 180,E1 -5499.323,E2 -5499.323} C_VEL
LIN {X 0,Y 510.07,Z 821.558,A -85,B 0,C 180,E1 -5500.419,E2 -5500.419} C_VEL
LIN {X 0,Y 510.388,Z 810.519,A -85,B 0,C 180,E1 -5501.417,E2 -5501.417} C_VEL
LIN {X 0,Y 510.662,Z 798.583,A -85,B 0,C 180,E1 -5502.274,E2 -5502.274} C_VEL
LIN {X 0,Y 510.972,Z 786.203,A -85,B 0,C 180,E1 -5502.966,E2 -5502.966} C_VEL
LIN {X 0,Y 511.315,Z 773.188,A -85,B 0,C 180,E1 -5503.513,E2 -5503.513} C_VEL
LIN {X 0,Y 511.573,Z 760.324,A -85,B 0,C 180,E1 -5503.886,E2 -5503.886} C_VEL
LIN {X 0,Y 511.79,Z 739.506,A -85,B 0,C 180,E1 -5504.235,E2 -5504.235} C_VEL
LIN {X 0,Y 512.103,Z 661.841,A -85,B 0,C 180,E1 -5505.353,E2 -5505.353} C_VEL
LIN {X 0,Y 510.511,Z 650.518,A -85,B 0,C 180,E1 -5505.57,E2 -5505.57} C_VEL
LIN {X 0,Y 510.248,Z 645.304,A -85,B 0,C 180,E1 -5505.682,E2 -5505.682} C_VEL
LIN {X 0,Y 510.559,Z 623.849,A -85,B 0,C 180,E1 -5508.666,E2 -5508.666} C_VEL
LIN {X 0,Y 510.754,Z 602.712,A -85,B 0,C 180,E1 -5511.598,E2 -5511.598} C_VEL
LIN {X 0,Y 510.9,Z 581.437,A -85,B 0,C 180,E1 -5514.577,E2 -5514.577} C_VEL
LIN {X 0,Y 511.004,Z 562.879,A -85,B 0,C 180,E1 -5517.213,E2 -5517.213} C_VEL
LIN {X 0,Y 511.029,Z 544.006,A -85,B 0,C 180,E1 -5519.955,E2 -5519.955} C_VEL
LIN {X 0,Y 509.95,Z 536.968,A -85,B 0,C 180,E1 -5521.045,E2 -5521.045} C_VEL
LIN {X 0,Y 509.864,Z 536.973,A -85,B 0,C 180,E1 -5524.203,E2 -5524.203} C_VEL
LIN {X 0,Y 509.821,Z 536.978,A -85,B 0,C 180,E1 -5527.341,E2 -5527.341} C_VEL
LIN {X 0,Y 509.842,Z 536.975,A -85,B 0,C 180,E1 -5530.382,E2 -5530.382} C_VEL
LIN {X 0,Y 509.827,Z 536.98,A -85,B 0,C 180,E1 -5533.062,E2 -5533.062} C_VEL
LIN {X 0,Y 509.835,Z 536.974,A -85,B 0,C 180,E1 -5535.792,E2 -5535.792} C_VEL
LIN {X 0,Y 509.863,Z 536.976,A -85,B 0,C 180,E1 -5538.575,E2 -5538.575} C_VEL
LIN {X 0,Y 509.856,Z 536.971,A -85,B 0,C 180,E1 -5541.786,E2 -5541.786} C_VEL
LIN {X 0,Y 509.834,Z 536.98,A -85,B 0,C 180,E1 -5544.622,E2 -5544.622} C_VEL
LIN {X 0,Y 509.866,Z 536.97,A -85,B 0,C 180,E1 -5547.481,E2 -5547.481} C_VEL
LIN {X 0,Y 509.863,Z 536.975,A -85,B 0,C 180,E1 -5550.274,E2 -5550.274} C_VEL
LIN {X 0,Y 509.89,Z 536.972,A -85,B 0,C 180,E1 -5552.944,E2 -5552.944} C_VEL
LIN {X 0,Y 509.875,Z 536.971,A -85,B 0,C 180,E1 -5555.574,E2 -5555.574} C_VEL
LIN {X 0,Y 509.855,Z 536.975,A -85,B 0,C 180,E1 -5558.998,E2 -5558.998} C_VEL
LIN {X 0,Y 509.886,Z 536.974,A -85,B 0,C 180,E1 -5562.001,E2 -5562.001} C_VEL
LIN {X 0,Y 509.91,Z 537.094,A -85,B 0,C 180,E1 -5563.308,E2 -5563.308} C_VEL
LIN {X 0,Y 513.209,Z 547.055,A -85,B 0,C 180,E1 -5563.55,E2 -5563.55} C_VEL
LIN {X 0,Y 513.18,Z 580.076,A -85,B 0,C 180,E1 -5564.031,E2 -5564.031} C_VEL
LIN {X 0,Y 513.097,Z 595.015,A -85,B 0,C 180,E1 -5564.406,E2 -5564.406} C_VEL
LIN {X 0,Y 512.945,Z 608.995,A -85,B 0,C 180,E1 -5564.91,E2 -5564.91} C_VEL
LIN {X 0,Y 512.64,Z 623.583,A -85,B 0,C 180,E1 -5565.612,E2 -5565.612} C_VEL
LIN {X 0,Y 512.287,Z 636.7,A -85,B 0,C 180,E1 -5566.412,E2 -5566.412} C_VEL
LIN {X 0,Y 511.965,Z 648.706,A -85,B 0,C 180,E1 -5567.312,E2 -5567.312} C_VEL
LIN {X 0,Y 511.553,Z 659.769,A -85,B 0,C 180,E1 -5568.308,E2 -5568.308} C_VEL
LIN {X 0,Y 511.085,Z 670.866,A -85,B 0,C 180,E1 -5569.502,E2 -5569.502} C_VEL
LIN {X 0,Y 510.718,Z 680.118,A -85,B 0,C 180,E1 -5570.695,E2 -5570.695} C_VEL
LIN {X 0,Y 510.384,Z 689.132,A -85,B 0,C 180,E1 -5572.085,E2 -5572.085} C_VEL
LIN {X 0,Y 510.195,Z 695.599,A -85,B 0,C 180,E1 -5573.276,E2 -5573.276} C_VEL
LIN {X 0,Y 509.876,Z 702.708,A -85,B 0,C 180,E1 -5574.859,E2 -5574.859} C_VEL
LIN {X 0,Y 509.678,Z 708.301,A -85,B 0,C 180,E1 -5576.442,E2 -5576.442} C_VEL
LIN {X 0,Y 509.53,Z 711.6,A -85,B 0,C 180,E1 -5577.628,E2 -5577.628} C_VEL
LIN {X 0,Y 509.454,Z 714.89,A -85,B 0,C 180,E1 -5579.209,E2 -5579.209} C_VEL
LIN {X 0,Y 509.438,Z 717.012,A -85,B 0,C 180,E1 -5580.79,E2 -5580.79} C_VEL
LIN {X 0,Y 509.481,Z 718.007,A -85,B 0,C 180,E1 -5582.371,E2 -5582.371} C_VEL
LIN {X 0,Y 509.429,Z 717.91,A -85,B 0,C 180,E1 -5583.955,E2 -5583.955} C_VEL
LIN {X 0,Y 509.454,Z 716.655,A -85,B 0,C 180,E1 -5585.541,E2 -5585.541} C_VEL
LIN {X 0,Y 509.521,Z 714.242,A -85,B 0,C 180,E1 -5587.131,E2 -5587.131} C_VEL
LIN {X 0,Y 509.6,Z 710.632,A -85,B 0,C 180,E1 -5588.725,E2 -5588.725} C_VEL
LIN {X 0,Y 509.659,Z 705.73,A -85,B 0,C 180,E1 -5590.327,E2 -5590.327} C_VEL
LIN {X 0,Y 509.923,Z 699.367,A -85,B 0,C 180,E1 -5591.931,E2 -5591.931} C_VEL
LIN {X 0,Y 510.194,Z 692.452,A -85,B 0,C 180,E1 -5593.34,E2 -5593.34} C_VEL
LIN {X 0,Y 510.508,Z 684.059,A -85,B 0,C 180,E1 -5594.754,E2 -5594.754} C_VEL
LIN {X 0,Y 510.922,Z 673.864,A -85,B 0,C 180,E1 -5596.173,E2 -5596.173} C_VEL
LIN {X 0,Y 511.355,Z 663.328,A -85,B 0,C 180,E1 -5597.393,E2 -5597.393} C_VEL
LIN {X 0,Y 511.826,Z 651.873,A -85,B 0,C 180,E1 -5598.502,E2 -5598.502} C_VEL
LIN {X 0,Y 512.245,Z 638.994,A -85,B 0,C 180,E1 -5599.537,E2 -5599.537} C_VEL
LIN {X 0,Y 512.667,Z 626.597,A -85,B 0,C 180,E1 -5600.356,E2 -5600.356} C_VEL
LIN {X 0,Y 513.072,Z 613.117,A -85,B 0,C 180,E1 -5601.075,E2 -5601.075} C_VEL
LIN {X 0,Y 513.433,Z 598.183,A -85,B 0,C 180,E1 -5601.689,E2 -5601.689} C_VEL
LIN {X 0,Y 513.578,Z 583.715,A -85,B 0,C 180,E1 -5602.127,E2 -5602.127} C_VEL
LIN {X 0,Y 513.683,Z 567.501,A -85,B 0,C 180,E1 -5602.439,E2 -5602.439} C_VEL
LIN {X 0,Y 513.645,Z 547.589,A -85,B 0,C 180,E1 -5602.735,E2 -5602.735} C_VEL
LIN {X 0,Y 509.842,Z 536.976,A -85,B 0,C 180,E1 -5603.048,E2 -5603.048} C_VEL
LIN {X 0,Y 509.913,Z 536.967,A -85,B 0,C 180,E1 -5606.378,E2 -5606.378} C_VEL
LIN {X 0,Y 509.878,Z 536.968,A -85,B 0,C 180,E1 -5608.844,E2 -5608.844} C_VEL
LIN {X 0,Y 509.821,Z 536.976,A -85,B 0,C 180,E1 -5611.59,E2 -5611.59} C_VEL
LIN {X 0,Y 509.848,Z 536.975,A -85,B 0,C 180,E1 -5614.413,E2 -5614.413} C_VEL
LIN {X 0,Y 509.818,Z 536.974,A -85,B 0,C 180,E1 -5617.34,E2 -5617.34} C_VEL
LIN {X 0,Y 509.84,Z 536.979,A -85,B 0,C 180,E1 -5620.382,E2 -5620.382} C_VEL
LIN {X 0,Y 509.824,Z 536.974,A -85,B 0,C 180,E1 -5623.062,E2 -5623.062} C_VEL
LIN {X 0,Y 509.824,Z 536.98,A -85,B 0,C 180,E1 -5624.303,E2 -5624.303} C_VEL
LIN {X 0,Y 509.159,Z 537.06,A -85,B 0,C 180,E1 -5624.962,E2 -5624.962} C_VEL
LIN {X 0,Y 506.277,Z 537.42,A -85,B 0,C 180,E1 -5626.033,E2 -5626.033} C_VEL
LIN {X 0,Y 503.861,Z 537.718,A -85,B 0,C 180,E1 -5626.895,E2 -5626.895} C_VEL
LIN {X 0,Y 502.862,Z 537.841,A -85,B 0,C 180,E1 -5627.562,E2 -5627.562} C_VEL
LIN {X 0,Y 502.801,Z 537.85,A -85,B 0,C 180,E1 -5627.787,E2 -5627.787} C_VEL
LIN {X 0,Y 502.789,Z 537.857,A -85,B 0,C 180,E1 -5630.245,E2 -5630.245} C_VEL
LIN {X 0,Y 502.774,Z 537.853,A -85,B 0,C 180,E1 -5633.053,E2 -5633.053} C_VEL
LIN {X 0,Y 502.806,Z 537.85,A -85,B 0,C 180,E1 -5636.006,E2 -5636.006} C_VEL
LIN {X 0,Y 502.796,Z 537.854,A -85,B 0,C 180,E1 -5638.856,E2 -5638.856} C_VEL
LIN {X 0,Y 502.843,Z 537.843,A -85,B 0,C 180,E1 -5641.704,E2 -5641.704} C_VEL
LIN {X 0,Y 502.84,Z 537.848,A -85,B 0,C 180,E1 -5644.324,E2 -5644.324} C_VEL
LIN {X 0,Y 502.81,Z 537.849,A -85,B 0,C 180,E1 -5647.295,E2 -5647.295} C_VEL
LIN {X 0,Y 502.825,Z 537.849,A -85,B 0,C 180,E1 -5650.4,E2 -5650.4} C_VEL
LIN {X 0,Y 502.834,Z 537.852,A -85,B 0,C 180,E1 -5652.931,E2 -5652.931} C_VEL
LIN {X 0,Y 502.844,Z 537.845,A -85,B 0,C 180,E1 -5655.429,E2 -5655.429} C_VEL
LIN {X 0,Y 502.876,Z 537.845,A -85,B 0,C 180,E1 -5658.716,E2 -5658.716} C_VEL
LIN {X 0,Y 502.901,Z 537.836,A -85,B 0,C 180,E1 -5661.966,E2 -5661.966} C_VEL
LIN {X 0,Y 502.936,Z 537.833,A -85,B 0,C 180,E1 -5664.386,E2 -5664.386} C_VEL
LIN {X 0,Y 503.024,Z 537.823,A -85,B 0,C 180,E1 -5667.597,E2 -5667.597} C_VEL
LIN {X 0,Y 503.026,Z 537.82,A -85,B 0,C 180,E1 -5670,E2 -5670} C_VEL
LIN {X 0,Y 503.024,Z 537.821,A -85,B 0,C 180,E1 -5672.402,E2 -5672.402} C_VEL
LIN {X 0,Y 502.932,Z 537.836,A -85,B 0,C 180,E1 -5675.613,E2 -5675.613} C_VEL
LIN {X 0,Y 502.899,Z 537.837,A -85,B 0,C 180,E1 -5678.033,E2 -5678.033} C_VEL
LIN {X 0,Y 502.89,Z 537.846,A -85,B 0,C 180,E1 -5681.282,E2 -5681.282} C_VEL
LIN {X 0,Y 502.842,Z 537.843,A -85,B 0,C 180,E1 -5684.57,E2 -5684.57} C_VEL
LIN {X 0,Y 502.859,Z 537.844,A -85,B 0,C 180,E1 -5687.906,E2 -5687.906} C_VEL
LIN {X 0,Y 502.825,Z 537.845,A -85,B 0,C 180,E1 -5690.536,E2 -5690.536} C_VEL
LIN {X 0,Y 502.793,Z 537.851,A -85,B 0,C 180,E1 -5693.04,E2 -5693.04} C_VEL
LIN {X 0,Y 502.838,Z 537.852,A -85,B 0,C 180,E1 -5695.675,E2 -5695.675} C_VEL
LIN {X 0,Y 502.839,Z 537.844,A -85,B 0,C 180,E1 -5698.372,E2 -5698.372} C_VEL
LIN {X 0,Y 502.794,Z 537.855,A -85,B 0,C 180,E1 -5701.5,E2 -5701.5} C_VEL
LIN {X 0,Y 502.803,Z 537.849,A -85,B 0,C 180,E1 -5704.445,E2 -5704.445} C_VEL
LIN {X 0,Y 502.776,Z 537.852,A -85,B 0,C 180,E1 -5707.178,E2 -5707.178} C_VEL
LIN {X 0,Y 502.817,Z 537.854,A -85,B 0,C 180,E1 -5710.012,E2 -5710.012} C_VEL
LIN {X 0,Y 502.768,Z 537.853,A -85,B 0,C 180,E1 -5713.231,E2 -5713.231} C_VEL
LIN {X 0,Y 502.785,Z 537.855,A -85,B 0,C 180,E1 -5715.661,E2 -5715.661} C_VEL
LIN {X 0,Y 502.824,Z 537.845,A -85,B 0,C 180,E1 -5718.935,E2 -5718.935} C_VEL
LIN {X 0,Y 502.792,Z 537.858,A -85,B 0,C 180,E1 -5722.046,E2 -5722.046} C_VEL
LIN {X 0,Y 502.805,Z 537.848,A -85,B 0,C 180,E1 -5725.035,E2 -5725.035} C_VEL
LIN {X 0,Y 502.784,Z 537.857,A -85,B 0,C 180,E1 -5727.916,E2 -5727.916} C_VEL
LIN {X 0,Y 502.866,Z 538.047,A -85,B 0,C 180,E1 -5729.202,E2 -5729.202} C_VEL
LIN {X 0,Y 506.173,Z 547.46,A -85,B 0,C 180,E1 -5729.459,E2 -5729.459} C_VEL
LIN {X 0,Y 505.842,Z 595.696,A -85,B 0,C 180,E1 -5730.19,E2 -5730.19} C_VEL
LIN {X 0,Y 505.626,Z 610.241,A -85,B 0,C 180,E1 -5730.577,E2 -5730.577} C_VEL
LIN {X 0,Y 505.449,Z 623.363,A -85,B 0,C 180,E1 -5731.088,E2 -5731.088} C_VEL
LIN {X 0,Y 505.079,Z 636.516,A -85,B 0,C 180,E1 -5731.765,E2 -5731.765} C_VEL
LIN {X 0,Y 504.694,Z 648.248,A -85,B 0,C 180,E1 -5732.531,E2 -5732.531} C_VEL
LIN {X 0,Y 504.308,Z 660.382,A -85,B 0,C 180,E1 -5733.516,E2 -5733.516} C_VEL
LIN {X 0,Y 503.825,Z 671.231,A -85,B 0,C 180,E1 -5734.591,E2 -5734.591} C_VEL
LIN {X 0,Y 503.456,Z 680.342,A -85,B 0,C 180,E1 -5735.682,E2 -5735.682} C_VEL
LIN {X 0,Y 503.142,Z 689.303,A -85,B 0,C 180,E1 -5736.977,E2 -5736.977} C_VEL
LIN {X 0,Y 502.884,Z 696.608,A -85,B 0,C 180,E1 -5738.263,E2 -5738.263} C_VEL
LIN {X 0,Y 502.664,Z 702.551,A -85,B 0,C 180,E1 -5739.541,E2 -5739.541} C_VEL
LIN {X 0,Y 502.503,Z 707.336,A -85,B 0,C 180,E1 -5740.812,E2 -5740.812} C_VEL
LIN {X 0,Y 502.455,Z 711.099,A -85,B 0,C 180,E1 -5742.078,E2 -5742.078} C_VEL
LIN {X 0,Y 502.322,Z 713.108,A -85,B 0,C 180,E1 -5742.914,E2 -5742.914} C_VEL
LIN {X 0,Y 502.258,Z 715.956,A -85,B 0,C 180,E1 -5744.582,E2 -5744.582} C_VEL
LIN {X 0,Y 502.26,Z 717.353,A -85,B 0,C 180,E1 -5746.239,E2 -5746.239} C_VEL
LIN {X 0,Y 502.279,Z 717.389,A -85,B 0,C 180,E1 -5747.885,E2 -5747.885} C_VEL
LIN {X 0,Y 502.279,Z 716.051,A -85,B 0,C 180,E1 -5749.52,E2 -5749.52} C_VEL
LIN {X 0,Y 502.335,Z 713.355,A -85,B 0,C 180,E1 -5751.148,E2 -5751.148} C_VEL
LIN {X 0,Y 502.545,Z 709.223,A -85,B 0,C 180,E1 -5752.77,E2 -5752.77} C_VEL
LIN {X 0,Y 502.669,Z 705.116,A -85,B 0,C 180,E1 -5753.981,E2 -5753.981} C_VEL
LIN {X 0,Y 502.771,Z 700.09,A -85,B 0,C 180,E1 -5755.189,E2 -5755.189} C_VEL
LIN {X 0,Y 503.042,Z 692.822,A -85,B 0,C 180,E1 -5756.596,E2 -5756.596} C_VEL
LIN {X 0,Y 503.308,Z 685.232,A -85,B 0,C 180,E1 -5757.8,E2 -5757.8} C_VEL
LIN {X 0,Y 503.749,Z 676.044,A -85,B 0,C 180,E1 -5759.001,E2 -5759.001} C_VEL
LIN {X 0,Y 504.064,Z 665.91,A -85,B 0,C 180,E1 -5760.1,E2 -5760.1} C_VEL
LIN {X 0,Y 504.526,Z 654.662,A -85,B 0,C 180,E1 -5761.098,E2 -5761.098} C_VEL
LIN {X 0,Y 504.975,Z 642.099,A -85,B 0,C 180,E1 -5761.994,E2 -5761.994} C_VEL
LIN {X 0,Y 505.312,Z 628.74,A -85,B 0,C 180,E1 -5762.741,E2 -5762.741} C_VEL
LIN {X 0,Y 505.558,Z 614.565,A -85,B 0,C 180,E1 -5763.338,E2 -5763.338} C_VEL
LIN {X 0,Y 505.724,Z 601.118,A -85,B 0,C 180,E1 -5763.735,E2 -5763.735} C_VEL
LIN {X 0,Y 505.777,Z 587.69,A -85,B 0,C 180,E1 -5763.984,E2 -5763.984} C_VEL
LIN {X 0,Y 506.054,Z 547.542,A -85,B 0,C 180,E1 -5764.556,E2 -5764.556} C_VEL
LIN {X 0,Y 502.87,Z 537.845,A -85,B 0,C 180,E1 -5764.811,E2 -5764.811} C_VEL
LIN {X 0,Y 502.929,Z 537.841,A -85,B 0,C 180,E1 -5767.225,E2 -5767.225} C_VEL
LIN {X 0,Y 502.819,Z 537.849,A -85,B 0,C 180,E1 -5770.469,E2 -5770.469} C_VEL
LIN {X 0,Y 502.828,Z 537.85,A -85,B 0,C 180,E1 -5772.923,E2 -5772.923} C_VEL
LIN {X 0,Y 502.845,Z 537.853,A -85,B 0,C 180,E1 -5775.4,E2 -5775.4} C_VEL
LIN {X 0,Y 502.843,Z 537.848,A -85,B 0,C 180,E1 -5778.123,E2 -5778.123} C_VEL
LIN {X 0,Y 502.826,Z 537.848,A -85,B 0,C 180,E1 -5780.537,E2 -5780.537} C_VEL
LIN {X 0,Y 502.794,Z 537.854,A -85,B 0,C 180,E1 -5783.041,E2 -5783.041} C_VEL
LIN {X 0,Y 502.84,Z 537.849,A -85,B 0,C 180,E1 -5785.676,E2 -5785.676} C_VEL
LIN {X 0,Y 502.839,Z 537.843,A -85,B 0,C 180,E1 -5788.373,E2 -5788.373} C_VEL
LIN {X 0,Y 502.795,Z 537.853,A -85,B 0,C 180,E1 -5791.5,E2 -5791.5} C_VEL
LIN {X 0,Y 502.801,Z 537.846,A -85,B 0,C 180,E1 -5794.445,E2 -5794.445} C_VEL
LIN {X 0,Y 502.777,Z 537.856,A -85,B 0,C 180,E1 -5797.179,E2 -5797.179} C_VEL
LIN {X 0,Y 502.787,Z 537.851,A -85,B 0,C 180,E1 -5800.016,E2 -5800.016} C_VEL
LIN {X 0,Y 502.802,Z 537.848,A -85,B 0,C 180,E1 -5802.2,E2 -5802.2} C_VEL
LIN {X 0,Y 502.8,Z 537.854,A -85,B 0,C 180,E1 -5805.469,E2 -5805.469} C_VEL
LIN {X 0,Y 502.819,Z 537.85,A -85,B 0,C 180,E1 -5808.935,E2 -5808.935} C_VEL
LIN {X 0,Y 502.794,Z 537.853,A -85,B 0,C 180,E1 -5812.047,E2 -5812.047} C_VEL
LIN {X 0,Y 502.809,Z 537.857,A -85,B 0,C 180,E1 -5815.036,E2 -5815.036} C_VEL
LIN {X 0,Y 502.877,Z 538.041,A -85,B 0,C 180,E1 -5816.593,E2 -5816.593} C_VEL
LIN {X 0,Y 505.764,Z 551.507,A -85,B 0,C 180,E1 -5819.06,E2 -5819.06} C_VEL
LIN {X 0,Y 505.645,Z 559.747,A -85,B 0,C 180,E1 -5820.435,E2 -5820.435} C_VEL
LIN {X 0,Y 505.025,Z 577.026,A -85,B 0,C 180,E1 -5823.241,E2 -5823.241} C_VEL
LIN {X 0,Y 504.413,Z 598.07,A -85,B 0,C 180,E1 -5826.58,E2 -5826.58} C_VEL
LIN {X 0,Y 503.905,Z 617.497,A -85,B 0,C 180,E1 -5829.594,E2 -5829.594} C_VEL
LIN {X 0,Y 503.438,Z 636.796,A -85,B 0,C 180,E1 -5832.535,E2 -5832.535} C_VEL
LIN {X 0,Y 503.212,Z 646.752,A -85,B 0,C 180,E1 -5834.036,E2 -5834.036} C_VEL
LIN {X 0,Y 505.495,Z 664.75,A -85,B 0,C 180,E1 -5834.418,E2 -5834.418} C_VEL
LIN {X 0,Y 505.041,Z 738.28,A -85,B 0,C 180,E1 -5835.494,E2 -5835.494} C_VEL
LIN {X 0,Y 504.791,Z 759.811,A -85,B 0,C 180,E1 -5835.873,E2 -5835.873} C_VEL
LIN {X 0,Y 504.505,Z 772.565,A -85,B 0,C 180,E1 -5836.25,E2 -5836.25} C_VEL
LIN {X 0,Y 504.051,Z 785.484,A -85,B 0,C 180,E1 -5836.803,E2 -5836.803} C_VEL
LIN {X 0,Y 503.76,Z 798.092,A -85,B 0,C 180,E1 -5837.527,E2 -5837.527} C_VEL
LIN {X 0,Y 503.429,Z 808.976,A -85,B 0,C 180,E1 -5838.322,E2 -5838.322} C_VEL
LIN {X 0,Y 503.029,Z 820.041,A -85,B 0,C 180,E1 -5839.332,E2 -5839.332} C_VEL
LIN {X 0,Y 502.76,Z 829.067,A -85,B 0,C 180,E1 -5840.344,E2 -5840.344} C_VEL
LIN {X 0,Y 502.544,Z 837.898,A -85,B 0,C 180,E1 -5841.557,E2 -5841.557} C_VEL
LIN {X 0,Y 502.347,Z 844.96,A -85,B 0,C 180,E1 -5842.767,E2 -5842.767} C_VEL
LIN {X 0,Y 502.306,Z 850.636,A -85,B 0,C 180,E1 -5843.977,E2 -5843.977} C_VEL
LIN {X 0,Y 502.146,Z 855.072,A -85,B 0,C 180,E1 -5845.183,E2 -5845.183} C_VEL
LIN {X 0,Y 502.232,Z 857.446,A -85,B 0,C 180,E1 -5845.988,E2 -5845.988} C_VEL
LIN {X 0,Y 502.154,Z 859.348,A -85,B 0,C 180,E1 -5846.791,E2 -5846.791} C_VEL
LIN {X 0,Y 502.143,Z 860.781,A -85,B 0,C 180,E1 -5847.594,E2 -5847.594} C_VEL
LIN {X 0,Y 502.039,Z 862.402,A -85,B 0,C 180,E1 -5849.198,E2 -5849.198} C_VEL
LIN {X 0,Y 502.061,Z 862.609,A -85,B 0,C 180,E1 -5850,E2 -5850} C_VEL
LIN {X 0,Y 502.081,Z 861.739,A -85,B 0,C 180,E1 -5851.605,E2 -5851.605} C_VEL
LIN {X 0,Y 502.15,Z 860.709,A -85,B 0,C 180,E1 -5852.407,E2 -5852.407} C_VEL
LIN {X 0,Y 502.164,Z 859.236,A -85,B 0,C 180,E1 -5853.21,E2 -5853.21} C_VEL
LIN {X 0,Y 502.201,Z 856.176,A -85,B 0,C 180,E1 -5854.415,E2 -5854.415} C_VEL
LIN {X 0,Y 502.287,Z 852.037,A -85,B 0,C 180,E1 -5855.621,E2 -5855.621} C_VEL
LIN {X 0,Y 502.357,Z 845.76,A -85,B 0,C 180,E1 -5857.012,E2 -5857.012} C_VEL
LIN {X 0,Y 502.532,Z 838.707,A -85,B 0,C 180,E1 -5858.242,E2 -5858.242} C_VEL
LIN {X 0,Y 502.734,Z 830.051,A -85,B 0,C 180,E1 -5859.455,E2 -5859.455} C_VEL
LIN {X 0,Y 503.02,Z 820.184,A -85,B 0,C 180,E1 -5860.567,E2 -5860.567} C_VEL
LIN {X 0,Y 503.37,Z 809.061,A -85,B 0,C 180,E1 -5861.578,E2 -5861.578} C_VEL
LIN {X 0,Y 503.635,Z 797.762,A -85,B 0,C 180,E1 -5862.402,E2 -5862.402} C_VEL
LIN {X 0,Y 503.964,Z 785.61,A -85,B 0,C 180,E1 -5863.098,E2 -5863.098} C_VEL
LIN {X 0,Y 504.327,Z 772.834,A -85,B 0,C 180,E1 -5863.653,E2 -5863.653} C_VEL
LIN {X 0,Y 504.636,Z 759.671,A -85,B 0,C 180,E1 -5864.055,E2 -5864.055} C_VEL
LIN {X 0,Y 504.853,Z 742.72,A -85,B 0,C 180,E1 -5864.358,E2 -5864.358} C_VEL
LIN {X 0,Y 505.186,Z 662.282,A -85,B 0,C 180,E1 -5865.551,E2 -5865.551} C_VEL
LIN {X 0,Y 503.684,Z 650.999,A -85,B 0,C 180,E1 -5865.775,E2 -5865.775} C_VEL
LIN {X 0,Y 503.18,Z 643.031,A -85,B 0,C 180,E1 -5865.931,E2 -5865.931} C_VEL
LIN {X 0,Y 503.467,Z 623.197,A -85,B 0,C 180,E1 -5868.728,E2 -5868.728} C_VEL
LIN {X 0,Y 503.658,Z 603.648,A -85,B 0,C 180,E1 -5871.487,E2 -5871.487} C_VEL
LIN {X 0,Y 503.835,Z 583.865,A -85,B 0,C 180,E1 -5874.299,E2 -5874.299} C_VEL
LIN {X 0,Y 503.949,Z 563.583,A -85,B 0,C 180,E1 -5877.23,E2 -5877.23} C_VEL
LIN {X 0,Y 503.998,Z 545.525,A -85,B 0,C 180,E1 -5879.902,E2 -5879.902} C_VEL
LIN {X 0,Y 502.91,Z 537.844,A -85,B 0,C 180,E1 -5881.107,E2 -5881.107} C_VEL
LIN {X 0,Y 502.808,Z 537.854,A -85,B 0,C 180,E1 -5884.444,E2 -5884.444} C_VEL
LIN {X 0,Y 502.782,Z 537.857,A -85,B 0,C 180,E1 -5887.178,E2 -5887.178} C_VEL
LIN {X 0,Y 502.792,Z 537.851,A -85,B 0,C 180,E1 -5890.015,E2 -5890.015} C_VEL
LIN {X 0,Y 502.807,Z 537.85,A -85,B 0,C 180,E1 -5892.199,E2 -5892.199} C_VEL
LIN {X 0,Y 502.805,Z 537.85,A -85,B 0,C 180,E1 -5895.468,E2 -5895.468} C_VEL
LIN {X 0,Y 502.825,Z 537.853,A -85,B 0,C 180,E1 -5898.934,E2 -5898.934} C_VEL
LIN {X 0,Y 502.798,Z 537.852,A -85,B 0,C 180,E1 -5902.046,E2 -5902.046} C_VEL
LIN {X 0,Y 502.803,Z 537.854,A -85,B 0,C 180,E1 -5905.034,E2 -5905.034} C_VEL
LIN {X 0,Y 502.788,Z 537.853,A -85,B 0,C 180,E1 -5907.915,E2 -5907.915} C_VEL
LIN {X 0,Y 502.829,Z 537.853,A -85,B 0,C 180,E1 -5910.712,E2 -5910.712} C_VEL
LIN {X 0,Y 502.867,Z 537.844,A -85,B 0,C 180,E1 -5913.439,E2 -5913.439} C_VEL
LIN {X 0,Y 502.796,Z 537.856,A -85,B 0,C 180,E1 -5916.086,E2 -5916.086} C_VEL
LIN {X 0,Y 502.788,Z 537.858,A -85,B 0,C 180,E1 -5918.689,E2 -5918.689} C_VEL
LIN {X 0,Y 502.833,Z 537.849,A -85,B 0,C 180,E1 -5921.248,E2 -5921.248} C_VEL
LIN {X 0,Y 502.854,Z 537.849,A -85,B 0,C 180,E1 -5923.074,E2 -5923.074} C_VEL
LIN {X 0,Y 506.4,Z 548.471,A -85,B 0,C 180,E1 -5923.353,E2 -5923.353} C_VEL
LIN {X 0,Y 506.33,Z 581.164,A -85,B 0,C 180,E1 -5923.831,E2 -5923.831} C_VEL
LIN {X 0,Y 506.287,Z 596.026,A -85,B 0,C 180,E1 -5924.205,E2 -5924.205} C_VEL
LIN {X 0,Y 506.153,Z 610.961,A -85,B 0,C 180,E1 -5924.755,E2 -5924.755} C_VEL
LIN {X 0,Y 505.843,Z 624.556,A -85,B 0,C 180,E1 -5925.414,E2 -5925.414} C_VEL
LIN {X 0,Y 505.462,Z 637.758,A -85,B 0,C 180,E1 -5926.225,E2 -5926.225} C_VEL
LIN {X 0,Y 505.103,Z 650.99,A -85,B 0,C 180,E1 -5927.239,E2 -5927.239} C_VEL
LIN {X 0,Y 504.662,Z 662.895,A -85,B 0,C 180,E1 -5928.35,E2 -5928.35} C_VEL
LIN {X 0,Y 504.123,Z 673.675,A -85,B 0,C 180,E1 -5929.558,E2 -5929.558} C_VEL
LIN {X 0,Y 503.82,Z 682.687,A -85,B 0,C 180,E1 -5930.768,E2 -5930.768} C_VEL
LIN {X 0,Y 503.424,Z 691.58,A -85,B 0,C 180,E1 -5932.197,E2 -5932.197} C_VEL
LIN {X 0,Y 503.147,Z 698.684,A -85,B 0,C 180,E1 -5933.584,E2 -5933.584} C_VEL
LIN {X 0,Y 502.853,Z 705.392,A -85,B 0,C 180,E1 -5935.189,E2 -5935.189} C_VEL
LIN {X 0,Y 502.681,Z 710.606,A -85,B 0,C 180,E1 -5936.794,E2 -5936.794} C_VEL
LIN {X 0,Y 502.512,Z 714.501,A -85,B 0,C 180,E1 -5938.397,E2 -5938.397} C_VEL
LIN {X 0,Y 502.423,Z 717.177,A -85,B 0,C 180,E1 -5940,E2 -5940} C_VEL
LIN {X 0,Y 502.383,Z 718.706,A -85,B 0,C 180,E1 -5941.603,E2 -5941.603} C_VEL
LIN {X 0,Y 502.404,Z 719.113,A -85,B 0,C 180,E1 -5943.207,E2 -5943.207} C_VEL
LIN {X 0,Y 502.434,Z 718.403,A -85,B 0,C 180,E1 -5944.814,E2 -5944.814} C_VEL
LIN {X 0,Y 502.514,Z 716.3,A -85,B 0,C 180,E1 -5946.559,E2 -5946.559} C_VEL
LIN {X 0,Y 502.567,Z 712.522,A -85,B 0,C 180,E1 -5948.443,E2 -5948.443} C_VEL
LIN {X 0,Y 502.674,Z 707.896,A -85,B 0,C 180,E1 -5950.065,E2 -5950.065} C_VEL
LIN {X 0,Y 502.904,Z 702.479,A -85,B 0,C 180,E1 -5951.535,E2 -5951.535} C_VEL
LIN {X 0,Y 503.168,Z 695.226,A -85,B 0,C 180,E1 -5953.118,E2 -5953.118} C_VEL
LIN {X 0,Y 503.521,Z 687.169,A -85,B 0,C 180,E1 -5954.55,E2 -5954.55} C_VEL
LIN {X 0,Y 503.934,Z 677.537,A -85,B 0,C 180,E1 -5955.972,E2 -5955.972} C_VEL
LIN {X 0,Y 504.347,Z 667.356,A -85,B 0,C 180,E1 -5957.224,E2 -5957.224} C_VEL
LIN {X 0,Y 504.829,Z 656.339,A -85,B 0,C 180,E1 -5958.359,E2 -5958.359} C_VEL
LIN {X 0,Y 505.256,Z 644.289,A -85,B 0,C 180,E1 -5959.399,E2 -5959.399} C_VEL
LIN {X 0,Y 505.764,Z 631.205,A -85,B 0,C 180,E1 -5960.328,E2 -5960.328} C_VEL
LIN {X 0,Y 506.196,Z 617.607,A -85,B 0,C 180,E1 -5961.107,E2 -5961.107} C_VEL
LIN {X 0,Y 506.575,Z 602.961,A -85,B 0,C 180,E1 -5961.762,E2 -5961.762} C_VEL
LIN {X 0,Y 506.73,Z 588.081,A -85,B 0,C 180,E1 -5962.257,E2 -5962.257} C_VEL
LIN {X 0,Y 506.902,Z 573.455,A -85,B 0,C 180,E1 -5962.581,E2 -5962.581} C_VEL
LIN {X 0,Y 506.883,Z 549.12,A -85,B 0,C 180,E1 -5962.959,E2 -5962.959} C_VEL
LIN {X 0,Y 502.794,Z 537.855,A -85,B 0,C 180,E1 -5963.29,E2 -5963.29} C_VEL
LIN {X 0,Y 502.866,Z 537.844,A -85,B 0,C 180,E1 -5966.566,E2 -5966.566} C_VEL
LIN {X 0,Y 502.826,Z 537.847,A -85,B 0,C 180,E1 -5969.287,E2 -5969.287} C_VEL
LIN {X 0,Y 502.784,Z 537.86,A -85,B 0,C 180,E1 -5972.084,E2 -5972.084} C_VEL
LIN {X 0,Y 502.8,Z 537.849,A -85,B 0,C 180,E1 -5974.965,E2 -5974.965} C_VEL
LIN {X 0,Y 502.794,Z 537.855,A -85,B 0,C 180,E1 -5977.953,E2 -5977.953} C_VEL
LIN {X 0,Y 502.821,Z 537.846,A -85,B 0,C 180,E1 -5981.065,E2 -5981.065} C_VEL
LIN {X 0,Y 502.786,Z 537.856,A -85,B 0,C 180,E1 -5984.53,E2 -5984.53} C_VEL
LIN {X 0,Y 502.801,Z 537.85,A -85,B 0,C 180,E1 -5987.787,E2 -5987.787} C_VEL
LIN {X 0,Y 502.194,Z 537.932,A -85,B 0,C 180,E1 -5988.456,E2 -5988.456} C_VEL
LIN {X 0,Y 499.366,Z 538.282,A -85,B 0,C 180,E1 -5989.542,E2 -5989.542} C_VEL
LIN {X 0,Y 496.925,Z 538.59,A -85,B 0,C 180,E1 -5990.417,E2 -5990.417} C_VEL
LIN {X 0,Y 495.854,Z 538.715,A -85,B 0,C 180,E1 -5991.093,E2 -5991.093} C_VEL
LIN {X 0,Y 495.756,Z 538.726,A -85,B 0,C 180,E1 -5991.322,E2 -5991.322} C_VEL
LIN {X 0,Y 495.751,Z 538.736,A -85,B 0,C 180,E1 -5994.462,E2 -5994.462} C_VEL
LIN {X 0,Y 495.768,Z 538.725,A -85,B 0,C 180,E1 -5997.405,E2 -5997.405} C_VEL
LIN {X 0,Y 495.766,Z 538.729,A -85,B 0,C 180,E1 -6000.253,E2 -6000.253} C_VEL
LIN {X 0,Y 495.823,Z 538.719,A -85,B 0,C 180,E1 -6003.25,E2 -6003.25} C_VEL
LIN {X 0,Y 495.752,Z 538.726,A -85,B 0,C 180,E1 -6005.725,E2 -6005.725} C_VEL
LIN {X 0,Y 495.743,Z 538.731,A -85,B 0,C 180,E1 -6008.371,E2 -6008.371} C_VEL
LIN {X 0,Y 495.784,Z 538.729,A -85,B 0,C 180,E1 -6010.971,E2 -6010.971} C_VEL
LIN {X 0,Y 495.779,Z 538.724,A -85,B 0,C 180,E1 -6013.53,E2 -6013.53} C_VEL
LIN {X 0,Y 495.796,Z 538.721,A -85,B 0,C 180,E1 -6016.055,E2 -6016.055} C_VEL
LIN {X 0,Y 495.85,Z 538.718,A -85,B 0,C 180,E1 -6018.554,E2 -6018.554} C_VEL
LIN {X 0,Y 495.872,Z 538.712,A -85,B 0,C 180,E1 -6021.852,E2 -6021.852} C_VEL
LIN {X 0,Y 495.894,Z 538.709,A -85,B 0,C 180,E1 -6024.306,E2 -6024.306} C_VEL
LIN {X 0,Y 495.993,Z 538.699,A -85,B 0,C 180,E1 -6027.563,E2 -6027.563} C_VEL
LIN {X 0,Y 495.997,Z 538.696,A -85,B 0,C 180,E1 -6030,E2 -6030} C_VEL
LIN {X 0,Y 495.992,Z 538.697,A -85,B 0,C 180,E1 -6032.436,E2 -6032.436} C_VEL
LIN {X 0,Y 495.888,Z 538.712,A -85,B 0,C 180,E1 -6035.693,E2 -6035.693} C_VEL
LIN {X 0,Y 495.87,Z 538.712,A -85,B 0,C 180,E1 -6038.147,E2 -6038.147} C_VEL
LIN {X 0,Y 495.865,Z 538.72,A -85,B 0,C 180,E1 -6041.444,E2 -6041.444} C_VEL
LIN {X 0,Y 495.787,Z 538.723,A -85,B 0,C 180,E1 -6044.782,E2 -6044.782} C_VEL
LIN {X 0,Y 495.786,Z 538.729,A -85,B 0,C 180,E1 -6047.318,E2 -6047.318} C_VEL
LIN {X 0,Y 495.775,Z 538.727,A -85,B 0,C 180,E1 -6049.89,E2 -6049.89} C_VEL
LIN {X 0,Y 495.762,Z 538.726,A -85,B 0,C 180,E1 -6052.862,E2 -6052.862} C_VEL
LIN {X 0,Y 495.796,Z 538.724,A -85,B 0,C 180,E1 -6056.067,E2 -6056.067} C_VEL
LIN {X 0,Y 495.776,Z 538.724,A -85,B 0,C 180,E1 -6058.814,E2 -6058.814} C_VEL
LIN {X 0,Y 495.756,Z 538.736,A -85,B 0,C 180,E1 -6061.726,E2 -6061.726} C_VEL
LIN {X 0,Y 495.773,Z 538.724,A -85,B 0,C 180,E1 -6064.695,E2 -6064.695} C_VEL
LIN {X 0,Y 495.727,Z 538.735,A -85,B 0,C 180,E1 -6067.561,E2 -6067.561} C_VEL
LIN {X 0,Y 495.775,Z 538.724,A -85,B 0,C 180,E1 -6070.698,E2 -6070.698} C_VEL
LIN {X 0,Y 495.729,Z 538.738,A -85,B 0,C 180,E1 -6074.001,E2 -6074.001} C_VEL
LIN {X 0,Y 495.757,Z 538.726,A -85,B 0,C 180,E1 -6077.121,E2 -6077.121} C_VEL
LIN {X 0,Y 495.789,Z 538.727,A -85,B 0,C 180,E1 -6080.366,E2 -6080.366} C_VEL
LIN {X 0,Y 495.73,Z 538.73,A -85,B 0,C 180,E1 -6083.457,E2 -6083.457} C_VEL
LIN {X 0,Y 495.756,Z 538.732,A -85,B 0,C 180,E1 -6086.436,E2 -6086.436} C_VEL
LIN {X 0,Y 495.765,Z 538.731,A -85,B 0,C 180,E1 -6088.956,E2 -6088.956} C_VEL
LIN {X 0,Y 499.397,Z 549.096,A -85,B 0,C 180,E1 -6089.25,E2 -6089.25} C_VEL
LIN {X 0,Y 499.041,Z 595.527,A -85,B 0,C 180,E1 -6089.96,E2 -6089.96} C_VEL
LIN {X 0,Y 498.842,Z 610.168,A -85,B 0,C 180,E1 -6090.343,E2 -6090.343} C_VEL
LIN {X 0,Y 498.665,Z 622.821,A -85,B 0,C 180,E1 -6090.828,E2 -6090.828} C_VEL
LIN {X 0,Y 498.315,Z 635.417,A -85,B 0,C 180,E1 -6091.461,E2 -6091.461} C_VEL
LIN {X 0,Y 497.905,Z 647.598,A -85,B 0,C 180,E1 -6092.238,E2 -6092.238} C_VEL
LIN {X 0,Y 497.527,Z 658.849,A -85,B 0,C 180,E1 -6093.127,E2 -6093.127} C_VEL
LIN {X 0,Y 497.071,Z 669.34,A -85,B 0,C 180,E1 -6094.129,E2 -6094.129} C_VEL
LIN {X 0,Y 496.623,Z 679.635,A -85,B 0,C 180,E1 -6095.325,E2 -6095.325} C_VEL
LIN {X 0,Y 496.222,Z 688.889,A -85,B 0,C 180,E1 -6096.637,E2 -6096.637} C_VEL
LIN {X 0,Y 495.964,Z 696.453,A -85,B 0,C 180,E1 -6097.944,E2 -6097.944} C_VEL
LIN {X 0,Y 495.668,Z 703.119,A -85,B 0,C 180,E1 -6099.356,E2 -6099.356} C_VEL
LIN {X 0,Y 495.499,Z 709.055,A -85,B 0,C 180,E1 -6100.961,E2 -6100.961} C_VEL
LIN {X 0,Y 495.435,Z 711.745,A -85,B 0,C 180,E1 -6101.882,E2 -6101.882} C_VEL
LIN {X 0,Y 495.259,Z 715.357,A -85,B 0,C 180,E1 -6103.513,E2 -6103.513} C_VEL
LIN {X 0,Y 495.246,Z 717.642,A -85,B 0,C 180,E1 -6105.201,E2 -6105.201} C_VEL
LIN {X 0,Y 495.238,Z 718.531,A -85,B 0,C 180,E1 -6106.876,E2 -6106.876} C_VEL
LIN {X 0,Y 495.297,Z 718.049,A -85,B 0,C 180,E1 -6108.542,E2 -6108.542} C_VEL
LIN {X 0,Y 495.308,Z 716.193,A -85,B 0,C 180,E1 -6110.197,E2 -6110.197} C_VEL
LIN {X 0,Y 495.415,Z 712.939,A -85,B 0,C 180,E1 -6111.845,E2 -6111.845} C_VEL
LIN {X 0,Y 495.627,Z 708.211,A -85,B 0,C 180,E1 -6113.487,E2 -6113.487} C_VEL
LIN {X 0,Y 495.747,Z 703.62,A -85,B 0,C 180,E1 -6114.713,E2 -6114.713} C_VEL
LIN {X 0,Y 496.027,Z 696.963,A -85,B 0,C 180,E1 -6116.141,E2 -6116.141} C_VEL
LIN {X 0,Y 496.314,Z 688.721,A -85,B 0,C 180,E1 -6117.566,E2 -6117.566} C_VEL
LIN {X 0,Y 496.731,Z 680.046,A -85,B 0,C 180,E1 -6118.784,E2 -6118.784} C_VEL
LIN {X 0,Y 497.018,Z 671.419,A -85,B 0,C 180,E1 -6119.798,E2 -6119.798} C_VEL
LIN {X 0,Y 497.499,Z 661.085,A -85,B 0,C 180,E1 -6120.81,E2 -6120.81} C_VEL
LIN {X 0,Y 497.877,Z 649.835,A -85,B 0,C 180,E1 -6121.719,E2 -6121.719} C_VEL
LIN {X 0,Y 498.303,Z 637.347,A -85,B 0,C 180,E1 -6122.526,E2 -6122.526} C_VEL
LIN {X 0,Y 498.584,Z 624.381,A -85,B 0,C 180,E1 -6123.182,E2 -6123.182} C_VEL
LIN {X 0,Y 498.81,Z 610.2,A -85,B 0,C 180,E1 -6123.711,E2 -6123.711} C_VEL
LIN {X 0,Y 498.887,Z 596.07,A -85,B 0,C 180,E1 -6124.065,E2 -6124.065} C_VEL
LIN {X 0,Y 499.1,Z 548.593,A -85,B 0,C 180,E1 -6124.77,E2 -6124.77} C_VEL
LIN {X 0,Y 495.847,Z 538.721,A -85,B 0,C 180,E1 -6125.032,E2 -6125.032} C_VEL
LIN {X 0,Y 495.901,Z 538.716,A -85,B 0,C 180,E1 -6127.328,E2 -6127.328} C_VEL
LIN {X 0,Y 495.796,Z 538.729,A -85,B 0,C 180,E1 -6129.794,E2 -6129.794} C_VEL
LIN {X 0,Y 495.848,Z 538.72,A -85,B 0,C 180,E1 -6132.275,E2 -6132.275} C_VEL
LIN {X 0,Y 495.804,Z 538.731,A -85,B 0,C 180,E1 -6135.624,E2 -6135.624} C_VEL
LIN {X 0,Y 495.803,Z 538.724,A -85,B 0,C 180,E1 -6138.248,E2 -6138.248} C_VEL
LIN {X 0,Y 495.771,Z 538.727,A -85,B 0,C 180,E1 -6140.757,E2 -6140.757} C_VEL
LIN {X 0,Y 495.75,Z 538.734,A -85,B 0,C 180,E1 -6143.387,E2 -6143.387} C_VEL
LIN {X 0,Y 495.797,Z 538.723,A -85,B 0,C 180,E1 -6146.068,E2 -6146.068} C_VEL
LIN {X 0,Y 495.776,Z 538.724,A -85,B 0,C 180,E1 -6148.815,E2 -6148.815} C_VEL
LIN {X 0,Y 495.757,Z 538.726,A -85,B 0,C 180,E1 -6151.727,E2 -6151.727} C_VEL
LIN {X 0,Y 495.77,Z 538.723,A -85,B 0,C 180,E1 -6154.695,E2 -6154.695} C_VEL
LIN {X 0,Y 495.729,Z 538.734,A -85,B 0,C 180,E1 -6157.562,E2 -6157.562} C_VEL
LIN {X 0,Y 495.766,Z 538.728,A -85,B 0,C 180,E1 -6160.7,E2 -6160.7} C_VEL
LIN {X 0,Y 495.734,Z 538.732,A -85,B 0,C 180,E1 -6163.696,E2 -6163.696} C_VEL
LIN {X 0,Y 495.728,Z 538.73,A -85,B 0,C 180,E1 -6166.306,E2 -6166.306} C_VEL
LIN {X 0,Y 495.766,Z 538.73,A -85,B 0,C 180,E1 -6169.301,E2 -6169.301} C_VEL
LIN {X 0,Y 495.731,Z 538.734,A -85,B 0,C 180,E1 -6172.439,E2 -6172.439} C_VEL
LIN {X 0,Y 495.785,Z 538.731,A -85,B 0,C 180,E1 -6175.458,E2 -6175.458} C_VEL
LIN {X 0,Y 495.804,Z 538.783,A -85,B 0,C 180,E1 -6176.318,E2 -6176.318} C_VEL
LIN {X 0,Y 498.856,Z 552.986,A -85,B 0,C 180,E1 -6178.959,E2 -6178.959} C_VEL
LIN {X 0,Y 498.773,Z 560.42,A -85,B 0,C 180,E1 -6180.219,E2 -6180.219} C_VEL
LIN {X 0,Y 498.058,Z 578.206,A -85,B 0,C 180,E1 -6183.158,E2 -6183.158} C_VEL
LIN {X 0,Y 497.458,Z 597.405,A -85,B 0,C 180,E1 -6186.257,E2 -6186.257} C_VEL
LIN {X 0,Y 496.877,Z 617.996,A -85,B 0,C 180,E1 -6189.509,E2 -6189.509} C_VEL
LIN {X 0,Y 496.371,Z 637.171,A -85,B 0,C 180,E1 -6192.49,E2 -6192.49} C_VEL
LIN {X 0,Y 496.176,Z 645.469,A -85,B 0,C 180,E1 -6193.759,E2 -6193.759} C_VEL
LIN {X 0,Y 498.723,Z 665.674,A -85,B 0,C 180,E1 -6194.201,E2 -6194.201} C_VEL
LIN {X 0,Y 498.293,Z 731.568,A -85,B 0,C 180,E1 -6195.189,E2 -6195.189} C_VEL
LIN {X 0,Y 497.91,Z 757.974,A -85,B 0,C 180,E1 -6195.648,E2 -6195.648} C_VEL
LIN {X 0,Y 497.571,Z 771.655,A -85,B 0,C 180,E1 -6196.055,E2 -6196.055} C_VEL
LIN {X 0,Y 497.134,Z 784.521,A -85,B 0,C 180,E1 -6196.615,E2 -6196.615} C_VEL
LIN {X 0,Y 496.75,Z 797.008,A -85,B 0,C 180,E1 -6197.343,E2 -6197.343} C_VEL
LIN {X 0,Y 496.441,Z 807.973,A -85,B 0,C 180,E1 -6198.155,E2 -6198.155} C_VEL
LIN {X 0,Y 496.008,Z 819.037,A -85,B 0,C 180,E1 -6199.18,E2 -6199.18} C_VEL
LIN {X 0,Y 495.706,Z 828.066,A -85,B 0,C 180,E1 -6200.205,E2 -6200.205} C_VEL
LIN {X 0,Y 495.487,Z 836.909,A -85,B 0,C 180,E1 -6201.435,E2 -6201.435} C_VEL
LIN {X 0,Y 495.276,Z 843.979,A -85,B 0,C 180,E1 -6202.663,E2 -6202.663} C_VEL
LIN {X 0,Y 495.25,Z 850.105,A -85,B 0,C 180,E1 -6203.999,E2 -6203.999} C_VEL
LIN {X 0,Y 495.121,Z 855.371,A -85,B 0,C 180,E1 -6205.523,E2 -6205.523} C_VEL
LIN {X 0,Y 495.108,Z 858.384,A -85,B 0,C 180,E1 -6206.746,E2 -6206.746} C_VEL
LIN {X 0,Y 495.097,Z 859.816,A -85,B 0,C 180,E1 -6207.56,E2 -6207.56} C_VEL
LIN {X 0,Y 495.038,Z 860.823,A -85,B 0,C 180,E1 -6208.373,E2 -6208.373} C_VEL
LIN {X 0,Y 495.005,Z 861.426,A -85,B 0,C 180,E1 -6209.187,E2 -6209.187} C_VEL
LIN {X 0,Y 495.054,Z 861.627,A -85,B 0,C 180,E1 -6210,E2 -6210} C_VEL
LIN {X 0,Y 495.049,Z 860.733,A -85,B 0,C 180,E1 -6211.628,E2 -6211.628} C_VEL
LIN {X 0,Y 495.112,Z 859.681,A -85,B 0,C 180,E1 -6212.441,E2 -6212.441} C_VEL
LIN {X 0,Y 495.126,Z 858.186,A -85,B 0,C 180,E1 -6213.255,E2 -6213.255} C_VEL
LIN {X 0,Y 495.157,Z 855.09,A -85,B 0,C 180,E1 -6214.478,E2 -6214.478} C_VEL
LIN {X 0,Y 495.228,Z 850.908,A -85,B 0,C 180,E1 -6215.702,E2 -6215.702} C_VEL
LIN {X 0,Y 495.313,Z 844.584,A -85,B 0,C 180,E1 -6217.112,E2 -6217.112} C_VEL
LIN {X 0,Y 495.476,Z 837.475,A -85,B 0,C 180,E1 -6218.36,E2 -6218.36} C_VEL
LIN {X 0,Y 495.67,Z 828.74,A -85,B 0,C 180,E1 -6219.591,E2 -6219.591} C_VEL
LIN {X 0,Y 495.934,Z 818.801,A -85,B 0,C 180,E1 -6220.72,E2 -6220.72} C_VEL
LIN {X 0,Y 496.369,Z 807.606,A -85,B 0,C 180,E1 -6221.744,E2 -6221.744} C_VEL
LIN {X 0,Y 496.64,Z 796.751,A -85,B 0,C 180,E1 -6222.546,E2 -6222.546} C_VEL
LIN {X 0,Y 496.95,Z 785.014,A -85,B 0,C 180,E1 -6223.234,E2 -6223.234} C_VEL
LIN {X 0,Y 497.39,Z 771.153,A -85,B 0,C 180,E1 -6223.847,E2 -6223.847} C_VEL
LIN {X 0,Y 497.683,Z 757.864,A -85,B 0,C 180,E1 -6224.256,E2 -6224.256} C_VEL
LIN {X 0,Y 497.94,Z 740.862,A -85,B 0,C 180,E1 -6224.561,E2 -6224.561} C_VEL
LIN {X 0,Y 498.364,Z 663.259,A -85,B 0,C 180,E1 -6225.745,E2 -6225.745} C_VEL
LIN {X 0,Y 496.889,Z 652.159,A -85,B 0,C 180,E1 -6225.974,E2 -6225.974} C_VEL
LIN {X 0,Y 496.128,Z 640.671,A -85,B 0,C 180,E1 -6226.2,E2 -6226.2} C_VEL
LIN {X 0,Y 496.425,Z 619.591,A -85,B 0,C 180,E1 -6229.218,E2 -6229.218} C_VEL
LIN {X 0,Y 496.614,Z 600.029,A -85,B 0,C 180,E1 -6232.026,E2 -6232.026} C_VEL
LIN {X 0,Y 496.741,Z 580.279,A -85,B 0,C 180,E1 -6234.892,E2 -6234.892} C_VEL
LIN {X 0,Y 496.881,Z 561.971,A -85,B 0,C 180,E1 -6237.595,E2 -6237.595} C_VEL
LIN {X 0,Y 496.901,Z 545.375,A -85,B 0,C 180,E1 -6240.104,E2 -6240.104} C_VEL
LIN {X 0,Y 495.853,Z 538.723,A -85,B 0,C 180,E1 -6241.184,E2 -6241.184} C_VEL
LIN {X 0,Y 495.786,Z 538.729,A -85,B 0,C 180,E1 -6244.543,E2 -6244.543} C_VEL
LIN {X 0,Y 495.734,Z 538.731,A -85,B 0,C 180,E1 -6247.562,E2 -6247.562} C_VEL
LIN {X 0,Y 495.771,Z 538.731,A -85,B 0,C 180,E1 -6250.7,E2 -6250.7} C_VEL
LIN {X 0,Y 495.738,Z 538.73,A -85,B 0,C 180,E1 -6254.001,E2 -6254.001} C_VEL
LIN {X 0,Y 495.731,Z 538.735,A -85,B 0,C 180,E1 -6257.117,E2 -6257.117} C_VEL
LIN {X 0,Y 495.764,Z 538.728,A -85,B 0,C 180,E1 -6259.953,E2 -6259.953} C_VEL
LIN {X 0,Y 495.733,Z 538.736,A -85,B 0,C 180,E1 -6262.553,E2 -6262.553} C_VEL
LIN {X 0,Y 495.782,Z 538.725,A -85,B 0,C 180,E1 -6265.457,E2 -6265.457} C_VEL
LIN {X 0,Y 495.76,Z 538.732,A -85,B 0,C 180,E1 -6268.364,E2 -6268.364} C_VEL
LIN {X 0,Y 495.792,Z 538.725,A -85,B 0,C 180,E1 -6271.507,E2 -6271.507} C_VEL
LIN {X 0,Y 495.796,Z 538.727,A -85,B 0,C 180,E1 -6273.932,E2 -6273.932} C_VEL
LIN {X 0,Y 495.766,Z 538.73,A -85,B 0,C 180,E1 -6277.139,E2 -6277.139} C_VEL
LIN {X 0,Y 495.776,Z 538.732,A -85,B 0,C 180,E1 -6280.109,E2 -6280.109} C_VEL
LIN {X 0,Y 495.803,Z 538.729,A -85,B 0,C 180,E1 -6282.837,E2 -6282.837} C_VEL
LIN {X 0,Y 499.651,Z 550.565,A -85,B 0,C 180,E1 -6283.152,E2 -6283.152} C_VEL
LIN {X 0,Y 499.548,Z 582.637,A -85,B 0,C 180,E1 -6283.629,E2 -6283.629} C_VEL
LIN {X 0,Y 499.479,Z 597.556,A -85,B 0,C 180,E1 -6284.01,E2 -6284.01} C_VEL
LIN {X 0,Y 499.354,Z 611.861,A -85,B 0,C 180,E1 -6284.542,E2 -6284.542} C_VEL
LIN {X 0,Y 499.037,Z 625.524,A -85,B 0,C 180,E1 -6285.211,E2 -6285.211} C_VEL
LIN {X 0,Y 498.643,Z 638.809,A -85,B 0,C 180,E1 -6286.033,E2 -6286.033} C_VEL
LIN {X 0,Y 498.274,Z 652.104,A -85,B 0,C 180,E1 -6287.061,E2 -6287.061} C_VEL
LIN {X 0,Y 497.852,Z 663.07,A -85,B 0,C 180,E1 -6288.085,E2 -6288.085} C_VEL
LIN {X 0,Y 497.239,Z 674.846,A -85,B 0,C 180,E1 -6289.412,E2 -6289.412} C_VEL
LIN {X 0,Y 496.93,Z 683.865,A -85,B 0,C 180,E1 -6290.639,E2 -6290.639} C_VEL
LIN {X 0,Y 496.513,Z 692.712,A -85,B 0,C 180,E1 -6292.08,E2 -6292.08} C_VEL
LIN {X 0,Y 496.193,Z 699.847,A -85,B 0,C 180,E1 -6293.493,E2 -6293.493} C_VEL
LIN {X 0,Y 495.873,Z 706.539,A -85,B 0,C 180,E1 -6295.121,E2 -6295.121} C_VEL
LIN {X 0,Y 495.689,Z 711.735,A -85,B 0,C 180,E1 -6296.748,E2 -6296.748} C_VEL
LIN {X 0,Y 495.511,Z 715.61,A -85,B 0,C 180,E1 -6298.374,E2 -6298.374} C_VEL
LIN {X 0,Y 495.414,Z 718.26,A -85,B 0,C 180,E1 -6300,E2 -6300} C_VEL
LIN {X 0,Y 495.368,Z 719.758,A -85,B 0,C 180,E1 -6301.626,E2 -6301.626} C_VEL
LIN {X 0,Y 495.376,Z 720.126,A -85,B 0,C 180,E1 -6303.253,E2 -6303.253} C_VEL
LIN {X 0,Y 495.423,Z 719.372,A -85,B 0,C 180,E1 -6304.882,E2 -6304.882} C_VEL
LIN {X 0,Y 495.509,Z 717.379,A -85,B 0,C 180,E1 -6306.556,E2 -6306.556} C_VEL
LIN {X 0,Y 495.515,Z 714.338,A -85,B 0,C 180,E1 -6308.154,E2 -6308.154} C_VEL
LIN {X 0,Y 495.686,Z 709.954,A -85,B 0,C 180,E1 -6309.796,E2 -6309.796} C_VEL
LIN {X 0,Y 495.909,Z 704.19,A -85,B 0,C 180,E1 -6311.443,E2 -6311.443} C_VEL
LIN {X 0,Y 496.192,Z 696.864,A -85,B 0,C 180,E1 -6313.098,E2 -6313.098} C_VEL
LIN {X 0,Y 496.54,Z 688.937,A -85,B 0,C 180,E1 -6314.55,E2 -6314.55} C_VEL
LIN {X 0,Y 496.961,Z 679.967,A -85,B 0,C 180,E1 -6315.918,E2 -6315.918} C_VEL
LIN {X 0,Y 497.426,Z 669.431,A -85,B 0,C 180,E1 -6317.259,E2 -6317.259} C_VEL
LIN {X 0,Y 497.907,Z 658.606,A -85,B 0,C 180,E1 -6318.41,E2 -6318.41} C_VEL
LIN {X 0,Y 498.372,Z 647.229,A -85,B 0,C 180,E1 -6319.428,E2 -6319.428} C_VEL
LIN {X 0,Y 498.888,Z 634.017,A -85,B 0,C 180,E1 -6320.405,E2 -6320.405} C_VEL
LIN {X 0,Y 499.334,Z 620.855,A -85,B 0,C 180,E1 -6321.195,E2 -6321.195} C_VEL
LIN {X 0,Y 499.701,Z 607.456,A -85,B 0,C 180,E1 -6321.835,E2 -6321.835} C_VEL
LIN {X 0,Y 499.934,Z 592.415,A -85,B 0,C 180,E1 -6322.38,E2 -6322.38} C_VEL
LIN {X 0,Y 500.123,Z 577.168,A -85,B 0,C 180,E1 -6322.756,E2 -6322.756} C_VEL
LIN {X 0,Y 500.14,Z 550.782,A -85,B 0,C 180,E1 -6323.176,E2 -6323.176} C_VEL
LIN {X 0,Y 495.759,Z 538.733,A -85,B 0,C 180,E1 -6323.532,E2 -6323.532} C_VEL
LIN {X 0,Y 495.816,Z 538.72,A -85,B 0,C 180,E1 -6326.974,E2 -6326.974} C_VEL
LIN {X 0,Y 495.766,Z 538.732,A -85,B 0,C 180,E1 -6330.147,E2 -6330.147} C_VEL
LIN {X 0,Y 495.794,Z 538.721,A -85,B 0,C 180,E1 -6333.244,E2 -6333.244} C_VEL
LIN {X 0,Y 495.721,Z 538.739,A -85,B 0,C 180,E1 -6336.088,E2 -6336.088} C_VEL
LIN {X 0,Y 495.765,Z 538.727,A -85,B 0,C 180,E1 -6338.768,E2 -6338.768} C_VEL
LIN {X 0,Y 495.758,Z 538.728,A -85,B 0,C 180,E1 -6341.78,E2 -6341.78} C_VEL
LIN {X 0,Y 495.737,Z 538.728,A -85,B 0,C 180,E1 -6345.14,E2 -6345.14} C_VEL
LIN {X 0,Y 495.757,Z 538.733,A -85,B 0,C 180,E1 -6348.218,E2 -6348.218} C_VEL
LIN {X 0,Y 495.756,Z 538.726,A -85,B 0,C 180,E1 -6351.322,E2 -6351.322} C_VEL
LIN {X 0,Y 495.06,Z 538.817,A -85,B 0,C 180,E1 -6352,E2 -6352} C_VEL
LIN {X 0,Y 492.197,Z 539.176,A -85,B 0,C 180,E1 -6353.102,E2 -6353.102} C_VEL
LIN {X 0,Y 489.805,Z 539.476,A -85,B 0,C 180,E1 -6353.99,E2 -6353.99} C_VEL
LIN {X 0,Y 488.794,Z 539.6,A -85,B 0,C 180,E1 -6354.675,E2 -6354.675} C_VEL
LIN {X 0,Y 488.72,Z 539.606,A -85,B 0,C 180,E1 -6354.907,E2 -6354.907} C_VEL
LIN {X 0,Y 488.703,Z 539.605,A -85,B 0,C 180,E1 -6357.853,E2 -6357.853} C_VEL
LIN {X 0,Y 488.723,Z 539.609,A -85,B 0,C 180,E1 -6360.729,E2 -6360.729} C_VEL
LIN {X 0,Y 488.756,Z 539.598,A -85,B 0,C 180,E1 -6363.528,E2 -6363.528} C_VEL
LIN {X 0,Y 488.693,Z 539.609,A -85,B 0,C 180,E1 -6366.254,E2 -6366.254} C_VEL
LIN {X 0,Y 488.745,Z 539.603,A -85,B 0,C 180,E1 -6369.175,E2 -6369.175} C_VEL
LIN {X 0,Y 488.758,Z 539.598,A -85,B 0,C 180,E1 -6371.627,E2 -6371.627} C_VEL
LIN {X 0,Y 488.761,Z 539.604,A -85,B 0,C 180,E1 -6374.999,E2 -6374.999} C_VEL
LIN {X 0,Y 488.804,Z 539.594,A -85,B 0,C 180,E1 -6378.387,E2 -6378.387} C_VEL
LIN {X 0,Y 488.816,Z 539.591,A -85,B 0,C 180,E1 -6381.733,E2 -6381.733} C_VEL
LIN {X 0,Y 488.853,Z 539.586,A -85,B 0,C 180,E1 -6384.224,E2 -6384.224} C_VEL
LIN {X 0,Y 488.96,Z 539.576,A -85,B 0,C 180,E1 -6387.528,E2 -6387.528} C_VEL
LIN {X 0,Y 488.952,Z 539.578,A -85,B 0,C 180,E1 -6390.823,E2 -6390.823} C_VEL
LIN {X 0,Y 488.96,Z 539.573,A -85,B 0,C 180,E1 -6392.471,E2 -6392.471} C_VEL
LIN {X 0,Y 488.846,Z 539.589,A -85,B 0,C 180,E1 -6395.775,E2 -6395.775} C_VEL
LIN {X 0,Y 488.815,Z 539.591,A -85,B 0,C 180,E1 -6398.266,E2 -6398.266} C_VEL
LIN {X 0,Y 488.827,Z 539.594,A -85,B 0,C 180,E1 -6401.611,E2 -6401.611} C_VEL
LIN {X 0,Y 488.759,Z 539.601,A -85,B 0,C 180,E1 -6405,E2 -6405} C_VEL
LIN {X 0,Y 488.751,Z 539.598,A -85,B 0,C 180,E1 -6408.442,E2 -6408.442} C_VEL
LIN {X 0,Y 488.703,Z 539.607,A -85,B 0,C 180,E1 -6411.07,E2 -6411.07} C_VEL
LIN {X 0,Y 488.69,Z 539.613,A -85,B 0,C 180,E1 -6413.745,E2 -6413.745} C_VEL
LIN {X 0,Y 488.795,Z 539.594,A -85,B 0,C 180,E1 -6416.945,E2 -6416.945} C_VEL
LIN {X 0,Y 488.715,Z 539.604,A -85,B 0,C 180,E1 -6420.365,E2 -6420.365} C_VEL
LIN {X 0,Y 488.732,Z 539.606,A -85,B 0,C 180,E1 -6423.484,E2 -6423.484} C_VEL
LIN {X 0,Y 488.685,Z 539.609,A -85,B 0,C 180,E1 -6426.356,E2 -6426.356} C_VEL
LIN {X 0,Y 488.737,Z 539.602,A -85,B 0,C 180,E1 -6429.25,E2 -6429.25} C_VEL
LIN {X 0,Y 488.707,Z 539.609,A -85,B 0,C 180,E1 -6431.6,E2 -6431.6} C_VEL
LIN {X 0,Y 488.706,Z 539.604,A -85,B 0,C 180,E1 -6434.801,E2 -6434.801} C_VEL
LIN {X 0,Y 488.726,Z 539.604,A -85,B 0,C 180,E1 -6437.479,E2 -6437.479} C_VEL
LIN {X 0,Y 488.764,Z 539.601,A -85,B 0,C 180,E1 -6439.68,E2 -6439.68} C_VEL
LIN {X 0,Y 488.679,Z 539.608,A -85,B 0,C 180,E1 -6442.842,E2 -6442.842} C_VEL
LIN {X 0,Y 488.73,Z 539.606,A -85,B 0,C 180,E1 -6445.888,E2 -6445.888} C_VEL
LIN {X 0,Y 488.741,Z 539.607,A -85,B 0,C 180,E1 -6448.715,E2 -6448.715} C_VEL
LIN {X 0,Y 492.576,Z 550.52,A -85,B 0,C 180,E1 -6449.03,E2 -6449.03} C_VEL
LIN {X 0,Y 492.215,Z 597.556,A -85,B 0,C 180,E1 -6449.769,E2 -6449.769} C_VEL
LIN {X 0,Y 492.006,Z 611.7,A -85,B 0,C 180,E1 -6450.153,E2 -6450.153} C_VEL
LIN {X 0,Y 491.797,Z 625.769,A -85,B 0,C 180,E1 -6450.714,E2 -6450.714} C_VEL
LIN {X 0,Y 491.415,Z 638.226,A -85,B 0,C 180,E1 -6451.374,E2 -6451.374} C_VEL
LIN {X 0,Y 490.993,Z 649.991,A -85,B 0,C 180,E1 -6452.159,E2 -6452.159} C_VEL
LIN {X 0,Y 490.547,Z 662.205,A -85,B 0,C 180,E1 -6453.174,E2 -6453.174} C_VEL
LIN {X 0,Y 490.048,Z 673.187,A -85,B 0,C 180,E1 -6454.29,E2 -6454.29} C_VEL
LIN {X 0,Y 489.636,Z 682.253,A -85,B 0,C 180,E1 -6455.402,E2 -6455.402} C_VEL
LIN {X 0,Y 489.245,Z 691.849,A -85,B 0,C 180,E1 -6456.831,E2 -6456.831} C_VEL
LIN {X 0,Y 488.904,Z 699.657,A -85,B 0,C 180,E1 -6458.275,E2 -6458.275} C_VEL
LIN {X 0,Y 488.63,Z 706.256,A -85,B 0,C 180,E1 -6459.807,E2 -6459.807} C_VEL
LIN {X 0,Y 488.484,Z 710.723,A -85,B 0,C 180,E1 -6461.113,E2 -6461.113} C_VEL
LIN {X 0,Y 488.347,Z 714.199,A -85,B 0,C 180,E1 -6462.409,E2 -6462.409} C_VEL
LIN {X 0,Y 488.227,Z 717.407,A -85,B 0,C 180,E1 -6464.128,E2 -6464.128} C_VEL
LIN {X 0,Y 488.201,Z 719.149,A -85,B 0,C 180,E1 -6465.835,E2 -6465.835} C_VEL
LIN {X 0,Y 488.25,Z 719.499,A -85,B 0,C 180,E1 -6467.531,E2 -6467.531} C_VEL
LIN {X 0,Y 488.248,Z 718.504,A -85,B 0,C 180,E1 -6469.215,E2 -6469.215} C_VEL
LIN {X 0,Y 488.324,Z 716.134,A -85,B 0,C 180,E1 -6470.891,E2 -6470.891} C_VEL
LIN {X 0,Y 488.498,Z 712.296,A -85,B 0,C 180,E1 -6472.561,E2 -6472.561} C_VEL
LIN {X 0,Y 488.699,Z 706.947,A -85,B 0,C 180,E1 -6474.223,E2 -6474.223} C_VEL
LIN {X 0,Y 488.849,Z 701.839,A -85,B 0,C 180,E1 -6475.465,E2 -6475.465} C_VEL
LIN {X 0,Y 489.167,Z 694.475,A -85,B 0,C 180,E1 -6476.912,E2 -6476.912} C_VEL
LIN {X 0,Y 489.515,Z 686.765,A -85,B 0,C 180,E1 -6478.149,E2 -6478.149} C_VEL
LIN {X 0,Y 490.014,Z 677.439,A -85,B 0,C 180,E1 -6479.384,E2 -6479.384} C_VEL
LIN {X 0,Y 490.388,Z 667.13,A -85,B 0,C 180,E1 -6480.514,E2 -6480.514} C_VEL
LIN {X 0,Y 490.883,Z 655.599,A -85,B 0,C 180,E1 -6481.539,E2 -6481.539} C_VEL
LIN {X 0,Y 491.311,Z 644.259,A -85,B 0,C 180,E1 -6482.357,E2 -6482.357} C_VEL
LIN {X 0,Y 491.64,Z 631.871,A -85,B 0,C 180,E1 -6483.073,E2 -6483.073} C_VEL
LIN {X 0,Y 491.914,Z 618.581,A -85,B 0,C 180,E1 -6483.661,E2 -6483.661} C_VEL
LIN {X 0,Y 492.045,Z 604.878,A -85,B 0,C 180,E1 -6484.096,E2 -6484.096} C_VEL
LIN {X 0,Y 492.085,Z 590.702,A -85,B 0,C 180,E1 -6484.377,E2 -6484.377} C_VEL
LIN {X 0,Y 492.274,Z 550.028,A -85,B 0,C 180,E1 -6484.98,E2 -6484.98} C_VEL
LIN {X 0,Y 488.827,Z 539.596,A -85,B 0,C 180,E1 -6485.277,E2 -6485.277} C_VEL
LIN {X 0,Y 488.814,Z 539.596,A -85,B 0,C 180,E1 -6488.267,E2 -6488.267} C_VEL
LIN {X 0,Y 488.826,Z 539.599,A -85,B 0,C 180,E1 -6491.612,E2 -6491.612} C_VEL
LIN {X 0,Y 488.759,Z 539.604,A -85,B 0,C 180,E1 -6495.001,E2 -6495.001} C_VEL
LIN {X 0,Y 488.752,Z 539.602,A -85,B 0,C 180,E1 -6498.443,E2 -6498.443} C_VEL
LIN {X 0,Y 488.704,Z 539.61,A -85,B 0,C 180,E1 -6501.071,E2 -6501.071} C_VEL
LIN {X 0,Y 488.691,Z 539.612,A -85,B 0,C 180,E1 -6503.746,E2 -6503.746} C_VEL
LIN {X 0,Y 488.797,Z 539.596,A -85,B 0,C 180,E1 -6506.946,E2 -6506.946} C_VEL
LIN {X 0,Y 488.717,Z 539.601,A -85,B 0,C 180,E1 -6510.365,E2 -6510.365} C_VEL
LIN {X 0,Y 488.733,Z 539.605,A -85,B 0,C 180,E1 -6513.485,E2 -6513.485} C_VEL
LIN {X 0,Y 488.682,Z 539.606,A -85,B 0,C 180,E1 -6516.355,E2 -6516.355} C_VEL
LIN {X 0,Y 488.7,Z 539.611,A -85,B 0,C 180,E1 -6519.255,E2 -6519.255} C_VEL
LIN {X 0,Y 488.722,Z 539.606,A -85,B 0,C 180,E1 -6521.603,E2 -6521.603} C_VEL
LIN {X 0,Y 488.711,Z 539.608,A -85,B 0,C 180,E1 -6524.802,E2 -6524.802} C_VEL
LIN {X 0,Y 488.691,Z 539.611,A -85,B 0,C 180,E1 -6527.475,E2 -6527.475} C_VEL
LIN {X 0,Y 488.732,Z 539.605,A -85,B 0,C 180,E1 -6529.677,E2 -6529.677} C_VEL
LIN {X 0,Y 488.682,Z 539.617,A -85,B 0,C 180,E1 -6532.842,E2 -6532.842} C_VEL
LIN {X 0,Y 488.738,Z 539.615,A -85,B 0,C 180,E1 -6536.052,E2 -6536.052} C_VEL
LIN {X 0,Y 491.93,Z 554.191,A -85,B 0,C 180,E1 -6538.81,E2 -6538.81} C_VEL
LIN {X 0,Y 491.992,Z 559.689,A -85,B 0,C 180,E1 -6539.766,E2 -6539.766} C_VEL
LIN {X 0,Y 491.15,Z 578.816,A -85,B 0,C 180,E1 -6542.979,E2 -6542.979} C_VEL
LIN {X 0,Y 490.474,Z 597.95,A -85,B 0,C 180,E1 -6546.122,E2 -6546.122} C_VEL
LIN {X 0,Y 489.86,Z 618.506,A -85,B 0,C 180,E1 -6549.421,E2 -6549.421} C_VEL
LIN {X 0,Y 489.254,Z 638.927,A -85,B 0,C 180,E1 -6552.659,E2 -6552.659} C_VEL
LIN {X 0,Y 489.081,Z 644.109,A -85,B 0,C 180,E1 -6553.466,E2 -6553.466} C_VEL
LIN {X 0,Y 491.937,Z 666.3,A -85,B 0,C 180,E1 -6553.966,E2 -6553.966} C_VEL
LIN {X 0,Y 491.446,Z 726.384,A -85,B 0,C 180,E1 -6554.898,E2 -6554.898} C_VEL
LIN {X 0,Y 491.011,Z 757.196,A -85,B 0,C 180,E1 -6555.442,E2 -6555.442} C_VEL
LIN {X 0,Y 490.658,Z 770.746,A -85,B 0,C 180,E1 -6555.854,E2 -6555.854} C_VEL
LIN {X 0,Y 490.208,Z 783.555,A -85,B 0,C 180,E1 -6556.423,E2 -6556.423} C_VEL
LIN {X 0,Y 489.759,Z 796.487,A -85,B 0,C 180,E1 -6557.191,E2 -6557.191} C_VEL
LIN {X 0,Y 489.394,Z 808.166,A -85,B 0,C 180,E1 -6558.087,E2 -6558.087} C_VEL
LIN {X 0,Y 488.998,Z 818.035,A -85,B 0,C 180,E1 -6559.023,E2 -6559.023} C_VEL
LIN {X 0,Y 488.653,Z 827.065,A -85,B 0,C 180,E1 -6560.062,E2 -6560.062} C_VEL
LIN {X 0,Y 488.414,Z 835.919,A -85,B 0,C 180,E1 -6561.31,E2 -6561.31} C_VEL
LIN {X 0,Y 488.22,Z 843.001,A -85,B 0,C 180,E1 -6562.557,E2 -6562.557} C_VEL
LIN {X 0,Y 488.191,Z 849.304,A -85,B 0,C 180,E1 -6563.955,E2 -6563.955} C_VEL
LIN {X 0,Y 488.065,Z 854.406,A -85,B 0,C 180,E1 -6565.458,E2 -6565.458} C_VEL
LIN {X 0,Y 488.063,Z 857.419,A -85,B 0,C 180,E1 -6566.698,E2 -6566.698} C_VEL
LIN {X 0,Y 488.051,Z 858.851,A -85,B 0,C 180,E1 -6567.525,E2 -6567.525} C_VEL
LIN {X 0,Y 488.001,Z 859.855,A -85,B 0,C 180,E1 -6568.35,E2 -6568.35} C_VEL
LIN {X 0,Y 488.045,Z 860.645,A -85,B 0,C 180,E1 -6570,E2 -6570} C_VEL
LIN {X 0,Y 488.017,Z 859.726,A -85,B 0,C 180,E1 -6571.651,E2 -6571.651} C_VEL
LIN {X 0,Y 488.074,Z 858.647,A -85,B 0,C 180,E1 -6572.476,E2 -6572.476} C_VEL
LIN {X 0,Y 488.089,Z 857.137,A -85,B 0,C 180,E1 -6573.302,E2 -6573.302} C_VEL
LIN {X 0,Y 488.119,Z 854.005,A -85,B 0,C 180,E1 -6574.542,E2 -6574.542} C_VEL
LIN {X 0,Y 488.172,Z 849.779,A -85,B 0,C 180,E1 -6575.784,E2 -6575.784} C_VEL
